// TIA Portal V18 program export: 0 tag tables, 0 data types, 166 data blocks, 119 code blocks (in call order from the OBs), 80 instance data blocks

DATA_BLOCK "GeneralDebug"   // DB1
{ S7_Optimized_Access := 'TRUE' }
// stored: MemoryReserve 100
   VAR
      Debug : Array[1..99] of Bool;
   END_VAR
BEGIN
END_DATA_BLOCK

DATA_BLOCK "DB_Commissioning"   // DB32767
{ S7_Optimized_Access := 'TRUE' }
// stored: AutoNumber false, MemoryReserve 100
   VAR RETAIN
      str : Array[1..8] of String[60];
      bit : Array[1..8] of Bool;
   END_VAR
BEGIN
   str[1] := 'LE4B171420124M33700000131950710';
END_DATA_BLOCK

DATA_BLOCK "DiagnosticDataBlock"   // DB3001
{ S7_Optimized_Access := 'FALSE' }
// stored: AutoNumber false
   VAR RETAIN
      DP : Struct
         DPReadStatus : Int;
         Status : Array[0..1023] of Bool;
      END_STRUCT;
      Profinet : Struct
         PNReadStatus : Int;
         Status : Array[0..1023] of Bool;
      END_STRUCT;
   END_VAR
BEGIN
   // DP.Status[0] : PLC-CPU
   // DP.Status[1] : Remote IO/ET200SP
   // DP.Status[2] : Festo Bus Coupler/总线耦合器
   // DP.Status[3] : CC-LINK
   // DP.Status[4] : Keyence Safety PLC
   // DP.Status[5] : Robot
   // DP.Status[6] : Keyence Laszer
   // DP.Status[7] : Balluff RFID
   // Profinet.Status[0] : ST70&ST80.PLC_CPU
   // Profinet.Status[1] : ST70&ST80.RFID
   // Profinet.Status[2] : ST70.Valves
   // Profinet.Status[3] : ST80.FCPN
   // Profinet.Status[4] : ST70.FCPN
   // Profinet.Status[5] : ST70.Screw
   // Profinet.Status[6] : CMMT-AS
   // Profinet.Status[7] : ST80.Screw
   // Profinet.Status[8] : ST80.Valves
END_DATA_BLOCK

DATA_BLOCK "Sys"   // DB3000
{ S7_Optimized_Access := 'FALSE' }
// stored: AutoNumber false
   VAR RETAIN
      COM : Struct   // Common
         AlwaysOFF : Bool := FALSE;
         AlwaysON : Bool := TRUE;
         FlashTime100mS : Bool := TRUE;   // Hardware Clock Memory 0.1S
         FlashTime200mS : Bool := TRUE;   // Hardware Clock Memory 0.2S
         FlashTime500mS : Bool := FALSE;   // Hardware Clock Memory 0.5S
         FlashTime1S : Bool := FALSE;   // Hardware Clock Memory 1S
         FlashTime2S : Bool := TRUE;   // Hardware Clock Memory 2S
         SpareBit : Bool := FALSE;
         PLCRestarted : Bool := TRUE;
      END_STRUCT;
      SpareB1 : Array[0..7] of Byte;
      DateTime : Struct   // DBX10.0
         Set : Date_And_Time := DT#1990-01-01-00:00:00;
         Read : Date_And_Time := DT#2025-03-12-08:03:05.785;
         Trigger : Bool := FALSE;   // Set
         ReturnValueRead : Int := 0;
         ReturnValueSet : Int := 0;
      END_STRUCT;
      SpareB2 : Array[0..17] of Byte;
      ScanTime : Struct   // DBX50.0
         CyclePrevious : Int := 14;
         CycleMax : Int := 23;
         CycleMin : Int := 9;
      END_STRUCT;
      RETVALI : Int := 0;
      RETVALW : Word := 16#0000;
      VersionManagement : Struct
         ProductLineName : String := 'Assembly Line';
         ProjectNumber : String[20] := 'SZ23055';
         "PLC IP Addr" : Array[0..3] of UInt;
         "HMI IP Addr" : Array[0..3] of UInt;
         PLCVersion : Array[0..1] of UInt;
         HMIVersion : Array[0..1] of UInt;
         "TIA Version" : String := 'TIA V18';
         StationID : Int := 10;
         HMIPageID : Int := 0;
      END_STRUCT;
   END_VAR
BEGIN
   SpareB1[0..7] := 16#00;
   SpareB2[0..17] := 16#00;
   VersionManagement."PLC IP Addr"[0] := 192;
   VersionManagement."PLC IP Addr"[1] := 168;
   VersionManagement."PLC IP Addr"[2..3] := 10;
   VersionManagement."HMI IP Addr"[0] := 192;
   VersionManagement."HMI IP Addr"[1] := 168;
   VersionManagement."HMI IP Addr"[2] := 45;
   VersionManagement."HMI IP Addr"[3] := 11;
   VersionManagement.PLCVersion[0] := 1;
   VersionManagement.PLCVersion[1] := 0;
   VersionManagement.HMIVersion[0] := 1;
   VersionManagement.HMIVersion[1] := 0;
END_DATA_BLOCK

DATA_BLOCK "ST10_GeneralData"   // DB1059
{ S7_Optimized_Access := 'FALSE' }
// stored: AutoNumber false
   VAR
      P_Plus : Array[0..50] of Bool;   // 脉冲沿信号使用Bool,使用需加注释
      ByPass : Array[0..10] of Bool;   // 屏蔽信号,使用需加注释
      HMI : Struct
         AREAPOINTER : Struct
            COORDINATION : Array[1..16] of Bool;
            USER_VERSION : Word;
            SCREEN_NUMBER : Struct
               SCREENTYPE : Int;
               SCREENNUMBER : Int;
               SPARE_1 : Int;
               FIELDNUMBER : Int;
               SPARE_2 : Int;
            END_STRUCT;
            JOB_MAILBOX : Struct
               JOBNUMBER : Int;
               PARAMETER_1 : Int;
               PARAMETER_2 : Int;
               PARAMETER_3 : Int;
            END_STRUCT;
            DATE_TIME_OP : Array[1..12] of Byte;
            DATE_TIME_PLC : Array[1..12] of Byte;
            SPARE : Array[1..22] of Byte;
            DataRecord : Struct   // 数据记录
               RecipeNummer : Word;
               DataRecordNummer : Word;
               Reserve : Word;
               TransferStatus : Word;   // 0,允许传送；2正在传送；4传送已完成，没有错误；12传送完成，出现错误
               Reserve_1 : Word;
            END_STRUCT;
         END_STRUCT;
         Win : Struct   // 弹窗相关变量
            Win : Int;
            WinBullfer : Int;
            "10x弹窗" : Array[1..10] of Int;
            "20x弹窗" : Array[1..10] of Int;
            "30x弹窗" : Array[1..10] of Int;
            "40x弹窗" : Array[1..10] of Int;
            TON : Array[1..40] of TON_TIME;
            "INT" { S7_SetPoint := 'True'} : Array[1..40] of Int;
            "Bool" : Array[1..40] of Bool;
         END_STRUCT;
         StationLightPB : Bool;   // 设备照明按钮
      END_STRUCT;
      Operator : Struct   // 操作员信息
         "Name" : String;   // 姓名
         ID : String;   // 工号
      END_STRUCT;
      TowerLamp : Struct
         PreReady : Bool;   // 等待托盘/等待人工操作
         PreStart : Bool;   // 人工操作完成（自动站False）
         ProcessingFinish : Bool;   // 加工完了 （单个产品加工完成）下个循环开始复位
         Maintenance : Bool;   // 维护提示（缺料OR保养置位1） 无---Flase
      END_STRUCT;
      FlowPartStatus { S7_SetPoint := 'True'} : Array[1..32] of Int;
      FunctionDeSelect : Struct   // 功能屏蔽选择
         "A" : Struct   // 单站屏蔽
            DeSelectPB_Servo380A1 : Bool;
            FunctionDeSelected_Servo380A1 : Bool;
            DeSelectPB_Servo381A1 : Bool;
            FunctionDeSelected_Servo381A1 : Bool;
            DeSelectPB_Servo383A1 : Bool;
            FunctionDeSelected_Servo383A1 : Bool;
            DeSelectPB_Reader800A1 : Bool;
            FunctionDeSelected_Reader800A1 : Bool;
            DeSelectPB_Reader801A1 : Bool;
            FunctionDeSelected_Reader801A1 : Bool;
            DeSelectPB_Reader802A1 : Bool;
            FunctionDeSelected_Reader802A1 : Bool;
            DeSelectPB_Reader803A1 : Bool;
            FunctionDeSelected_Reader803A1 : Bool;
            DeSelectPB_Reader804A1 : Bool;
            FunctionDeSelected_Reader804A1 : Bool;
         END_STRUCT;
         "B" : Struct   // RFID屏蔽
            DeSelectPB_Press372A1 : Bool;
            FunctionDeSelected_Press372A1 : Bool;
            DeSelectPB_Press375A1 : Bool;
            FunctionDeSelected_Press375A1 : Bool;
            DeSelectPB_Reader806A1 : Bool;
            FunctionDeSelected_Reader806A1 : Bool;
            DeSelectPB_TestPress372A1 : Bool;
            FunctionDeSelected_TestPress372A1 : Bool;
            DeSelectPB_TestPress375A1 : Bool;
            FunctionDeSelected_TestPress375A1 : Bool;
         END_STRUCT;
         C : Struct   // 扫码枪屏蔽
            DeSelectPB_Servo382A1 : Bool;
            FunctionDeSelected_Servo382A1 : Bool;
            DeSelectPB_ServoIAI : Bool;
            FunctionDeSelected_ServoIAI : Bool;
            DeSelectPB_IV3810A1 : Bool;
            FunctionDeSelected_IV3810A1 : Bool;
            DeSelectPB_IV3811A1 : Bool;
            FunctionDeSelected_IV3811A1 : Bool;
            DeSelectPB_Glue : Bool;
            FunctionDeSelected_Glue : Bool;
         END_STRUCT;
         "E" : Struct   // 注油屏蔽
            DeSelectPB : Bool;
            FunctionDeSelected : Bool;
         END_STRUCT;
         F : Struct   // 螺丝枪屏蔽
            DeSelectPB_Reader805A1 : Bool;
            FunctionDeSelected_Reader805A1 : Bool;
         END_STRUCT;
         H : Struct   // 油漆笔屏蔽
            DeSelectPB : Bool;
            FunctionDeSelected : Bool;
         END_STRUCT;
         J : Struct   // 油漆笔屏蔽
            DeSelectPB : Bool;
            FunctionDeSelected : Bool;
         END_STRUCT;
         K : Struct   // 油漆笔屏蔽
            DeSelectPB : Bool;
            FunctionDeSelected : Bool;
         END_STRUCT;
         L : Struct   // 油漆笔屏蔽
            DeSelectPB : Bool;
            FunctionDeSelected : Bool;
         END_STRUCT;
         MES : Struct   // MES屏蔽
            DeSelectPB : Bool;
            FunctionDeSelected : Bool;
         END_STRUCT;
         Global : Struct
            DeSelectPB_DryMode : Bool;
            FunctionDeSelected_DryMode : Bool;
            DeSelectPB_ScanFixture : Bool;
            FunctionDeSelected_ScanFixture : Bool;
            Spare_2 : Bool;
            Spare_3 : Bool;
            Spare_4 : Bool;
            Spare_5 : Bool;
            Spare_6 : Bool;
            Spare_7 : Bool;
            Spare_8 : Bool;
            Spare_9 : Bool;
            Spare_10 : Bool;
            Spare_11 : Bool;
            Spare_12 : Bool;
            Spare_13 : Bool;
         END_STRUCT;
      END_STRUCT;
      FlowControl_Handshake : Array[1..32] of Struct   // 流程控制的互锁
         PartPresent : Bool;
         initi : Bool;   // 初始化
         Start : Bool;
         Running : Bool;
         Done : Bool;
         Bypass : Bool;
      END_STRUCT;
      FixtureIDCheck { S7_SetPoint := 'True'} : Array[1..16] of "FixtureCheck_UDT";   // 工装匹配
      ProcessData { S7_SetPoint := 'True'} : Array[0..5] of "ProcessData";
   END_VAR
BEGIN
   // FlowControl_Handshake[2].Bypass : 流程NG
   // FlowControl_Handshake[1] : 主加工流程控制的互锁
   // FlowControl_Handshake[2] : 打标流程控制的互锁
   // FlowControl_Handshake[3] : 产品定位流程控制的互锁
   // FlowControl_Handshake[4] : 贴标流程控制互锁
END_DATA_BLOCK

DATA_BLOCK "Station_Sys"   // DB1060
TITLE = Station system DB
{ S7_Optimized_Access := 'FALSE' }
AUTHOR : RCS
FAMILY : Sys
VERSION : 2.0
// update 20160218
// stored: AutoNumber false
   VAR RETAIN
      ScreenNo : Int;   // For change HMI screen
      SpareB01 : Array[0..7] of Byte;   // *******************************************************************************
      Status : "RCS_SysStatus_V1";   // DBX10.0
      Input : Struct   // DBX20.0 For change PLC I input to PLC inside bit
         OP1 : Struct
            "Function 1" : Bool;
            "Function 2" : Bool;
            "Function 3" : Bool;
            "Function 4" : Bool;
            "Function 5" : Bool;
            "Function 6" : Bool;
            "Function 7" : Bool;
            "Function 8" : Bool;
         END_STRUCT;
         OP2 : Struct
            "Function 1" : Bool;
            "Function 2" : Bool;
            "Function 3" : Bool;
         END_STRUCT;
         OP3 : Struct
            "Function 1" : Bool;
            "Function 2" : Bool;
            "Function 3" : Bool;
         END_STRUCT;
      END_STRUCT;
      SpareB02 : Array[0..13] of Byte;   // *******************************************************************************
      HMI : Struct   // DBX40.0 HMI relation
         AP : Struct   // Area Pointer struct
            S1 : Int;
            CurrentScreenID : Int;
            S3 : Int;
            S4 : Int;
            S5 : Int;
         END_STRUCT;
      END_STRUCT;
      Cmd : "RCS_SysCmd_V1";   // DBX50.0
      SpareB03 : Array[0..7] of Byte;   // *******************************************************************************
      Interface : "RCS_SysComInterface_V1";   // DBX60.0
      SpareB04 : Array[0..3] of Byte;   // *******************************************************************************
      Initial : Struct   // DBX70.0
         Set : Bool;   // Trigger by HMI Button,[0]Total trigger
         Running : Bool;   // [0]Total initial Running
         OK : Bool;   // finish
      END_STRUCT;
      SpareB05 : Array[0..27] of Byte;   // *******************************************************************************
      Auto : "RCS_SysAuto_V1";   // DBX100.0
      SpareB10 : Array[0..5] of Byte;   // *******************************************************************************
      "A" : Struct   // DBX110.0 Auto control bit for some device
         "Device1 Auto control" : Bool;
         "Device2 Auto control" : Bool;
         "Device3 Auto control" : Bool;
         "Device4 Auto control" : Bool;
         "Device 01" : Struct
            "Function 1" : Bool;   // Flash
            "Function 2" : Bool;
            "Function 3" : Bool;   // Flash
         END_STRUCT;
         "Device 02" : Struct
            "Function 1" : Bool;   // Flash
            "Function 2" : Bool;
            "Function 3" : Bool;   // Flash
         END_STRUCT;
      END_STRUCT;
      SpareB11 : Array[0..33] of Byte;   // *******************************************************************************
      Manual : "RCS_SysManual_V1";   // DBX150.0
      SpareB12 : Array[0..6] of Byte;   // *******************************************************************************
      "M" : Struct   // DBX160.0 Manual control bit for some device
         "Device1 Manual control" : Bool;
         "Device2 Manual control" : Bool;
         "Device3 Manual control" : Bool;
         "Device4 Manual control" : Bool;
      END_STRUCT;
      SpareB13 : Array[0..37] of Byte;   // *******************************************************************************
      Safety : "RCS_SysSafety_V1";   // DBX200.0
      SpareB20 : Array[0..9] of Byte;   // *******************************************************************************
      Signal : Struct   // DBX220.0
         MainPressureSwitch1 : Bool;
         MainPressureSwitch2 : Bool;
         MainPressureSwitch3 : Bool;
      END_STRUCT;
      SpareB21 : Array[0..36] of Byte;   // *******************************************************************************
      Flag : Struct   // DBX260.0
         Processstart : Bool;
         PeocessComplete : Bool;
         IndexTable : Struct
            Interlock : Bool;
            TableRunning : Bool;   // Complete cycle Running
            StopandPosition : Bool;
            PositionOK : Bool;
            PositionNG : Bool;
            FixtureOK : Bool;
            FixtureNG : Bool;
            InitialOK : Bool;
         END_STRUCT;
      END_STRUCT;
      SpareB22 : Array[0..5] of Byte;   // *******************************************************************************
      P : Struct   // Positive RLO Edge Detection:-(P)- DBX270
         Record : Bool;
         "Set index run" : Bool;
         initial : Array[0..7] of Bool;
      END_STRUCT;
      SpareB23 : Array[0..5] of Byte;   // *******************************************************************************
      N : Struct   // Negative RLO Edge Detection:-(N)- DBX280
         Spare : Bool;
      END_STRUCT;
      SpareB24 : Array[0..17] of Byte;   // *******************************************************************************
      Alarm : "RCS_SysAlarmWarning_V1";   // DBX300.0
      SpareB30 : Array[0..7] of Byte;   // *******************************************************************************
      Warning : "RCS_SysAlarmWarning_V1";   // DBX310.0 / DBX500.0
      SpareB31 : Array[0..7] of Byte;   // *******************************************************************************
      AlarmTimes : Struct   // DBX320 If a fault continue happened over Limit times, than Auto running will be stopped / If a fault continue happened over Limit_times，Auto running will be stopped
         ForceStop : Bool;   // DBX320.0 / DBX650.0
         Reset : Bool;
         Limit : Int;
      END_STRUCT;
      SpareB33 : Array[0..5] of Byte;   // *******************************************************************************
      AlarmWarning : Int;   // DBX330 1:Alarm 2:Warning / DBX660 1:Alarm 2:Warning
      SpareB34 : Array[0..17] of Byte;   // *******************************************************************************
      Count : "RCS_SysCount_V1";   // DBX350.0 / DBX700.0
      SpareB40 : Array[0..11] of Byte;   // *******************************************************************************
      TotalCycleTime : "RCS_SysCycleTime_V1";   // DBX500.0 / DBX850.0
      SpareB41 : Array[0..11] of Byte;   // *******************************************************************************
      MachineCycleTime : "RCS_SysCycleTime_V1";   // DBX600.0 / DBX950.0
      SpareB42 : Array[0..11] of Byte;   // *******************************************************************************
      UserName { S7_SetPoint := 'True'} : String[20];   // DBX700.0
   END_VAR
BEGIN
   // Cmd.Record : 记录
   // Cmd.BuzzerOn : 蜂鸣器 On
   Cmd.OnOffLine := TRUE;
END_DATA_BLOCK

DATA_BLOCK "ST10_SysInput"   // DB1001
{ S7_Optimized_Access := 'TRUE' }
// stored: AutoNumber false, MemoryReserve 100
   VAR
      HMI_Button : Struct
         ControlOn : Bool := false;   // HMI_上电按钮
         ControlOff : Bool;   // HMI_断电按钮
         MachineStart : Bool := false;   // HMI_设备启动按钮
         MachineStop : Bool := false;   // HMI_设备停止按钮
         ResetButton : Bool := false;   // HMI_复位按钮
         "Manual/Auto" : Bool := false;   // HMI_手/自动切换按钮
         SafetyGateUnlock : Bool := false;   // HMI_安全门解锁按钮
         "E-Stop" : Bool := false;   // HMI_急停
      END_STRUCT;
      Sys : Struct
         iCircuitBreakerOK1 : Bool;   // 电子断路器 OK
         iCircuitBreakerOK2 : Bool;
         iPressure : Bool;   // 气压监控
      END_STRUCT;
      "iE-StopPB" : Array[1..20] of Bool;   // 急停按钮PB
      iSafetyGatFeedBack : Array[1..20] of Bool;   // 安全门
      iSafetydoorLockingFeedBack : Array[1..20] of Bool;   // 安全门反馈
      iMaterieldoorLockingFeedBack : Array[1..20] of Bool;   // 安全门反馈
   END_VAR
BEGIN
END_DATA_BLOCK

DATA_BLOCK "ST10_SysOutput"   // DB1002
{ S7_Optimized_Access := 'TRUE' }
// stored: AutoNumber false, MemoryReserve 100
   VAR
      oTowerLight : Struct
         Red : Bool;
         Yellow : Bool;
         Green : Bool;
         Blue : Bool;
      END_STRUCT;
      HMIButtonLight : Struct
         ControlOn : Bool := false;   // HMI_上电按钮
         ControlOff : Bool;   // HMI_断电按钮
         MachineStart : Bool := false;   // HMI_设备启动按钮
         MachineStop : Bool := false;   // HMI_设备停止按钮
         ResetButton : Bool := false;   // HMI_复位按钮
         "Manual/Auto" : Bool := false;   // HMI_手/自动切换按钮
         SafetyGateUnlock : Bool := false;   // HMI_安全门解锁按钮
      END_STRUCT;
      BoxLight : Struct
         oMachineStartLight : Bool;   // 启动按钮PB
         oMachineStopLight : Bool;   // 停止按钮PB
         oResetLight : Bool;   // 复位按钮PB
         oSafetyGateUnlockLight : Bool;   // 安全门解锁按钮PB
      END_STRUCT;
      SafetyDoorCoil : Array[1..20] of Bool;
      MaterialDoorCoil : Array[1..20] of Bool;
   END_VAR
BEGIN
END_DATA_BLOCK

DATA_BLOCK "AutoProcessControl"   // DB5100
{ S7_Optimized_Access := 'FALSE' }
// stored: AutoNumber false
   VAR
      A_Table_1Scan : Struct   // 自动页面
         Robot1PickPrimit : Bool;
         Spare_2 : Bool;
         Spare_3 : Bool;
         Spare_4 : Bool;
         Spare_5 : Bool;
         Spare_6 : Bool;
         Spare_7 : Bool;
         Spare_8 : Bool;
         Spare_9 : Bool;
         Spare_10 : Bool;
         Spare_11 : Bool;
         Spare_12 : Bool;
         Spare_13 : Bool;
         Spare_14 : Bool;
         Spare_15 : Bool;
         Spare_16 : Bool;
      END_STRUCT;
      A_Table_1Loading : Struct
         Robot1PickPrimit : Bool;
         Spare_2 : Bool;
         Spare_3 : Bool;
         Spare_4 : Bool;
         Spare_5 : Bool;
         Spare_6 : Bool;
         Spare_7 : Bool;
         Spare_8 : Bool;
         Spare_9 : Bool;
         Spare_10 : Bool;
         Spare_11 : Bool;
         Spare_12 : Bool;
         Spare_13 : Bool;
         Spare_14 : Bool;
         Spare_15 : Bool;
         Spare_16 : Bool;
         ServoRunCount : Int;
      END_STRUCT;
      A_Table_2Scan : Struct
         Robot3PickPrimit : Bool;
         Spare_2 : Bool;
         Spare_3 : Bool;
         Spare_4 : Bool;
         Spare_5 : Bool;
         Spare_6 : Bool;
         Spare_7 : Bool;
         Spare_8 : Bool;
         Spare_9 : Bool;
         Spare_10 : Bool;
         Spare_11 : Bool;
         Spare_12 : Bool;
         Spare_13 : Bool;
         Spare_14 : Bool;
         Spare_15 : Bool;
         Spare_16 : Bool;
      END_STRUCT;
      A_Table_2Loading : Struct
         Robot3PickPrimit : Bool;
         Spare_2 : Bool;
         Spare_3 : Bool;
         Spare_4 : Bool;
         Spare_5 : Bool;
         Spare_6 : Bool;
         Spare_7 : Bool;
         Spare_8 : Bool;
         Spare_9 : Bool;
         Spare_10 : Bool;
         Spare_11 : Bool;
         Spare_12 : Bool;
         Spare_13 : Bool;
         Spare_14 : Bool;
         Spare_15 : Bool;
         Spare_16 : Bool;
         ServoRunCount : Int;
      END_STRUCT;
      A_ScanRotary : Struct
         Robot1PickPrimit : Bool;
         Robot1PutPrimit : Bool;
         Spare_3 : Bool;
         Spare_4 : Bool;
         Spare_5 : Bool;
         Spare_6 : Bool;
         Spare_7 : Bool;
         Spare_8 : Bool;
         Spare_9 : Bool;
         Spare_10 : Bool;
         Spare_11 : Bool;
         Spare_12 : Bool;
         Spare_13 : Bool;
         Spare_14 : Bool;
         Spare_15 : Bool;
         Spare_16 : Bool;
      END_STRUCT;
      B_Press_1 : Struct   // 自动页面
         Robot1PickPrimit : Bool;
         Robot1PutShaftPrimit : Bool;
         Robot1PutRingPrimit : Bool;
         Spare_4 : Bool;
         Spare_5 : Bool;
         Spare_6 : Bool;
         Spare_7 : Bool;
         Spare_8 : Bool;
         Spare_9 : Bool;
         Spare_10 : Bool;
         Spare_11 : Bool;
         Spare_12 : Bool;
         Spare_13 : Bool;
         Spare_14 : Bool;
         Spare_15 : Bool;
         Spare_16 : Bool;
         GripStatus : Int;
      END_STRUCT;
      B_Press_2 : Struct
         Robot3PickPrimit : Bool;
         Robot3PutRingPrimit : Bool;
         Robot2PutPrimit : Bool;
         Spare_4 : Bool;
         Spare_5 : Bool;
         Spare_6 : Bool;
         Spare_7 : Bool;
         Spare_8 : Bool;
         Spare_9 : Bool;
         Spare_10 : Bool;
         Spare_11 : Bool;
         Spare_12 : Bool;
         Spare_13 : Bool;
         Spare_14 : Bool;
         Spare_15 : Bool;
         Spare_16 : Bool;
         GripStatus : Int;
      END_STRUCT;
      C_Glue : Struct
         Robot2PickPrimit : Bool;
         Robot1PutPrimit : Bool;
         Robot2MaganePutPrimit : Bool;
         Spare_4 : Bool;
         Spare_5 : Bool;
         Spare_6 : Bool;
         Spare_7 : Bool;
         Spare_8 : Bool;
         GlueTest : Bool;
         Spare_10 : Bool;
         Spare_11 : Bool;
         Spare_12 : Bool;
         Spare_13 : Bool;
         Spare_14 : Bool;
         Spare_15 : Bool;
         Spare_16 : Bool;
      END_STRUCT;
      H_ShafeLine : Struct
         Robot1PickPrimit : Bool;
         Spare_2 : Bool;
         Spare_3 : Bool;
         Spare_4 : Bool;
         Spare_5 : Bool;
         Spare_6 : Bool;
         Spare_7 : Bool;
         Spare_8 : Bool;
         EmptyMaterial : Bool;   // 托盘清料反转
         LineTest : Bool;
         Spare_11 : Bool;
         Spare_12 : Bool;
         Spare_13 : Bool;
         Spare_14 : Bool;
         Spare_15 : Bool;
         Spare_16 : Bool;
      END_STRUCT;
      J_MagnetLine : Struct
         Robot2PickPrimit : Bool;
         Spare_2 : Bool;
         Spare_3 : Bool;
         Spare_4 : Bool;
         Spare_5 : Bool;
         Spare_6 : Bool;
         Spare_7 : Bool;
         Spare_8 : Bool;
         EmptyMaterial : Bool;   // 托盘清料反转
         LineTest : Bool;
         Spare_11 : Bool;
         Spare_12 : Bool;
         Spare_13 : Bool;
         Spare_14 : Bool;
         Spare_15 : Bool;
         Spare_16 : Bool;
      END_STRUCT;
      K_ShafeLine : Struct
         Robot2PickPrimit : Bool;
         Spare_2 : Bool;
         Spare_3 : Bool;
         Spare_4 : Bool;
         Spare_5 : Bool;
         Spare_6 : Bool;
         Spare_7 : Bool;
         Spare_8 : Bool;
         EmptyMaterial : Bool;   // 托盘清料反转
         LineTest : Bool;
         Spare_11 : Bool;
         Spare_12 : Bool;
         Spare_13 : Bool;
         Spare_14 : Bool;
         Spare_15 : Bool;
         Spare_16 : Bool;
      END_STRUCT;
      L_ShafeLine : Struct
         Robot3PutPrimit : Bool;
         Spare_2 : Bool;
         Spare_3 : Bool;
         Spare_4 : Bool;
         Spare_5 : Bool;
         Spare_6 : Bool;
         Spare_7 : Bool;
         Spare_8 : Bool;
         EmptyMaterial : Bool;   // 托盘清料反转
         LineTest : Bool;
         Spare_11 : Bool;
         Spare_12 : Bool;
         Spare_13 : Bool;
         Spare_14 : Bool;
         Spare_15 : Bool;
         Spare_16 : Bool;
      END_STRUCT;
      Headt : Struct
         PalletUnloadingPrimit : Bool;
         Spare_2 : Bool;
         Spare_3 : Bool;
         Spare_4 : Bool;
         Spare_5 : Bool;
         Spare_6 : Bool;
         Spare_7 : Bool;
         Spare_8 : Bool;
         Spare_9 : Bool;
         Spare_10 : Bool;
         Spare_11 : Bool;
         Spare_12 : Bool;
         Spare_13 : Bool;
         Spare_14 : Bool;
         Spare_15 : Bool;
         Spare_16 : Bool;
      END_STRUCT;
      Robot2ScanNG : Struct
         PutPrimit : Bool;
         Spare_2 : Bool;
         Spare_3 : Bool;
         Spare_4 : Bool;
         Spare_5 : Bool;
         Spare_6 : Bool;
         Spare_7 : Bool;
         Spare_8 : Bool;
         Spare_9 : Bool;
         Spare_10 : Bool;
         Spare_11 : Bool;
         Spare_12 : Bool;
         Spare_13 : Bool;
         Spare_14 : Bool;
         Spare_15 : Bool;
         Spare_16 : Bool;
      END_STRUCT;
      Robot2GlueNG : Struct
         PutPrimit : Bool;
         Spare_2 : Bool;
         Spare_3 : Bool;
         Spare_4 : Bool;
         Spare_5 : Bool;
         Spare_6 : Bool;
         Spare_7 : Bool;
         Spare_8 : Bool;
         Spare_9 : Bool;
         Spare_10 : Bool;
         Spare_11 : Bool;
         Spare_12 : Bool;
         Spare_13 : Bool;
         Spare_14 : Bool;
         Spare_15 : Bool;
         Spare_16 : Bool;
      END_STRUCT;
      NG_1 : Struct
         Robot1PutPrimit_1 : Bool;
         Robot1PutPrimit_2 : Bool;
         Robot1PutPrimit_3 : Bool;
         Spare_4 : Bool;
         Spare_5 : Bool;
         Spare_6 : Bool;
         Spare_7 : Bool;
         Spare_8 : Bool;
         DoorRequest : Bool;
         Spare_10 : Bool;
         Spare_11 : Bool;
         Spare_12 : Bool;
         Spare_13 : Bool;
         Spare_14 : Bool;
         Spare_15 : Bool;
         Spare_16 : Bool;
      END_STRUCT;
      NG_2 : Struct
         Robot3PutPrimit_1 : Bool;
         Robot3PutPrimit_2 : Bool;
         Robot3PutPrimit_3 : Bool;
         Spare_4 : Bool;
         Spare_5 : Bool;
         Spare_6 : Bool;
         Spare_7 : Bool;
         Spare_8 : Bool;
         DoorRequest : Bool;
         Spare_10 : Bool;
         Spare_11 : Bool;
         Spare_12 : Bool;
         Spare_13 : Bool;
         Spare_14 : Bool;
         Spare_15 : Bool;
         Spare_16 : Bool;
      END_STRUCT;
      NGBuffer : Struct
         Robot3PPickMagnetNGPrimit : Bool;
         PickGlueNGPrimit : Bool;
         Spare_17 : Bool;
         Spare_4 : Bool;
         Spare_5 : Bool;
         Spare_6 : Bool;
         Spare_7 : Bool;
         Spare_8 : Bool;
         Spare_9 : Bool;
         Spare_10 : Bool;
         Spare_11 : Bool;
         Spare_12 : Bool;
         Spare_13 : Bool;
         Spare_14 : Bool;
         Spare_15 : Bool;
         Spare_16 : Bool;
      END_STRUCT;
      Fixture1Code : Struct
         Robot1CodeReadReq : Bool;
         Spare_17 : Bool;
         Spare_18 : Bool;
         Spare_4 : Bool;
         Spare_5 : Bool;
         Spare_6 : Bool;
         Spare_7 : Bool;
         Spare_8 : Bool;
         Spare_9 : Bool;
         Spare_10 : Bool;
         Spare_11 : Bool;
         Spare_12 : Bool;
         Spare_13 : Bool;
         Spare_14 : Bool;
         Spare_15 : Bool;
         Spare_16 : Bool;
      END_STRUCT;
      Fixture2Code : Struct
         Robot3CodeReadReq : Bool;
         Spare_17 : Bool;
         Spare_18 : Bool;
         Spare_4 : Bool;
         Spare_5 : Bool;
         Spare_6 : Bool;
         Spare_7 : Bool;
         Spare_8 : Bool;
         Spare_9 : Bool;
         Spare_10 : Bool;
         Spare_11 : Bool;
         Spare_12 : Bool;
         Spare_13 : Bool;
         Spare_14 : Bool;
         Spare_15 : Bool;
         Spare_16 : Bool;
      END_STRUCT;
      Robot_1 : Struct
         GluePutFlag : Bool;
         NGPutFlag : Bool;
         MaintenanceRequest : Bool;
         HomeRequest : Bool;
         Spare_5 : Bool;
         Spare_6 : Bool;
         Spare_7 : Bool;
         Spare_8 : Bool;
         ReadyToRobot2 : Bool;
         ClearPart : Bool;
         GripScanRequest : Bool;
         OnePart : Bool;
         Spare_13 : Bool;
         Spare_14 : Bool;
         Spare_15 : Bool;
         Spare_16 : Bool;
      END_STRUCT;
      Robot_2 : Struct
         PalletPickFlag : Bool;
         MagnetScanFlag : Bool;
         GluePutFlag : Bool;
         GluePickFlag : Bool;
         Press2PutFlag : Bool;
         GlueNGPutFlag : Bool;
         ScanNGPutFlag : Bool;
         Spare_8 : Bool;
         ReadyToRobot1 : Bool;
         ReadyToRobot3 : Bool;
         MaintenanceRequest : Bool;
         HomeRequest : Bool;
         GripScanRequest : Bool;
         Spare_14 : Bool;
         Spare_15 : Bool;
         Spare_16 : Bool;
      END_STRUCT;
      Robot_3 : Struct
         Press2PutFlag : Bool;
         Press2PickFlag : Bool;
         GlueNGPickFlag : Bool;
         ScanNGPickFlag : Bool;
         NGPutFlag : Bool;
         Spare_10 : Bool;
         Spare_9 : Bool;
         Spare_8 : Bool;
         ReadyToRobot2 : Bool;
         PalletFull : Bool;
         MaintenanceRequest : Bool;
         HomeRequest : Bool;
         GripScanRequest : Bool;
         Spare_14 : Bool;
         Spare_15 : Bool;
         Spare_16 : Bool;
      END_STRUCT;
      Global : Struct
         H : Struct
            EmptyPallet : Bool;
            LoadStopRequestPallet_1 : Bool;
            LoadStopRequestPallet_2 : Bool;
            LoadStopRequestPallet_3 : Bool;
            LoadStopRequestPallet_4 : Bool;
            EmptyStopRequestPallet_1 : Bool;
            EmptyStopRequestPallet_2 : Bool;
            EmptyStopRequestPallet_3 : Bool;
            Spare : Bool;
            Spare_1 : Bool;
            Spare_2 : Bool;
            Spare_3 : Bool;
            Spare_4 : Bool;
            Spare_5 : Bool;
            Spare_6 : Bool;
            Spare_7 : Bool;
         END_STRUCT;
         J : Struct
            EmptyPallet : Bool;
            LoadStopRequestPallet_1 : Bool;
            LoadStopRequestPallet_2 : Bool;
            LoadStopRequestPallet_3 : Bool;
            LoadStopRequestPallet_4 : Bool;
            EmptyStopRequestPallet_1 : Bool;
            EmptyStopRequestPallet_2 : Bool;
            EmptyStopRequestPallet_3 : Bool;
            Spare : Bool;
            Spare_1 : Bool;
            Spare_2 : Bool;
            Spare_3 : Bool;
            Spare_4 : Bool;
            Spare_5 : Bool;
            Spare_6 : Bool;
            Spare_7 : Bool;
         END_STRUCT;
         K : Struct
            EmptyPallet : Bool;
            LoadStopRequestPallet_1 : Bool;
            LoadStopRequestPallet_2 : Bool;
            LoadStopRequestPallet_3 : Bool;
            LoadStopRequestPallet_4 : Bool;
            EmptyStopRequestPallet_1 : Bool;
            EmptyStopRequestPallet_2 : Bool;
            EmptyStopRequestPallet_3 : Bool;
            Spare : Bool;
            Spare_1 : Bool;
            Spare_2 : Bool;
            Spare_3 : Bool;
            Spare_4 : Bool;
            Spare_5 : Bool;
            Spare_6 : Bool;
            Spare_7 : Bool;
         END_STRUCT;
         L : Struct
            EmptyPallet : Bool;
            LoadStopRequestPallet_1 : Bool;
            LoadStopRequestPallet_2 : Bool;
            LoadStopRequestPallet_3 : Bool;
            LoadStopRequestPallet_4 : Bool;
            EmptyStopRequestPallet_1 : Bool;
            EmptyStopRequestPallet_2 : Bool;
            EmptyStopRequestPallet_3 : Bool;
            Spare : Bool;
            Spare_1 : Bool;
            Spare_2 : Bool;
            Spare_3 : Bool;
            Spare_4 : Bool;
            Spare_5 : Bool;
            Spare_6 : Bool;
            Spare_7 : Bool;
         END_STRUCT;
         H_EmptyPallet : Bool;
         J_EmptyPallet : Bool;
         K_EmptyPallet : Bool;
         L_EmptyPallet : Bool;
         ALL_EmptyPallet : Bool;
         ALL_BeltPalletEmptyFinish : Bool;
         Spare_7 : Bool;
         Spare_8 : Bool;
         Spare_9 : Bool;
         Spare_10 : Bool;
         Spare_11 : Bool;
         Spare_12 : Bool;
         Spare_13 : Bool;
         Spare_14 : Bool;
         Spare_15 : Bool;
         Spare_16 : Bool;
         P : Array[0..60] of Bool;
      END_STRUCT;
      P : Array[0..40] of Bool;
      Status : Struct
         A1TableScan : Struct
            Status : Int;
         END_STRUCT;
         A1TableUnloading : Struct
            Status : Int;
         END_STRUCT;
         A1RotaryScan : Struct
            Status : Int;
         END_STRUCT;
         B1Press : Struct
            Status : Int;
         END_STRUCT;
         FRobot_1 : Struct
            Status : Int;
         END_STRUCT;
         A1FixtureCodeScan : Struct
            Status : Int;
         END_STRUCT;
         CGlueing : Struct
            Status : Int;
         END_STRUCT;
         FRobot_2 : Struct
            Status : Int;
         END_STRUCT;
         A2TableScan : Struct
            Status : Int;
         END_STRUCT;
         A2TableUnloading : Struct
            Status : Int;
         END_STRUCT;
         ChangeOver : Struct
            Status : Int;
         END_STRUCT;
         B2Press : Struct
            Status : Int;
         END_STRUCT;
         FRobot_3 : Struct
            Status : Int;
         END_STRUCT;
         A2FixtureCodeScan : Struct
            Status : Int;
         END_STRUCT;
         HShaftLifting : Struct
            Status : Int;
         END_STRUCT;
         JMagnetLifting : Struct
            Status : Int;
         END_STRUCT;
         KReserveLifting : Struct
            Status : Int;
         END_STRUCT;
         LUnloadingTrans : Struct
            Status : Int;
         END_STRUCT;
         "HShaftLoad&Unload" : Struct
            Status : Int;
         END_STRUCT;
         "JMagnetLoad&Unload" : Struct
            Status : Int;
         END_STRUCT;
         "KReserveLoad&Unload" : Struct
            Status : Int;
         END_STRUCT;
         "LUnloadingLoad&Unload" : Struct
            Status : Int;
         END_STRUCT;
         Solidify : Struct
            Status : Int;
         END_STRUCT;
         ENG_1 : Struct
            Status : Int;
         END_STRUCT;
         ENG_2 : Struct
            Status : Int;
         END_STRUCT;
      END_STRUCT;
   END_VAR
BEGIN
END_DATA_BLOCK

DATA_BLOCK "AutoProcessData"   // DB1600
{ S7_Optimized_Access := 'FALSE' }
// stored: AutoNumber false
   VAR RETAIN
      A_ScanRotate : "ProcessData";
      F_Robot1Grip1 { S7_SetPoint := 'True'} : "ProcessData";
      F_Robot1Grip2 { S7_SetPoint := 'True'} : "ProcessData";
      B_Press1 { S7_SetPoint := 'True'} : "ProcessData";
      C_Glue { S7_SetPoint := 'True'} : "ProcessData";
      F_Robot2Grip1 { S7_SetPoint := 'True'} : "ProcessData";
      F_Robot2Grip2 { S7_SetPoint := 'True'} : "ProcessData";
      C_GlueNGBuffer { S7_SetPoint := 'True'} : "ProcessData";
      C_MagnScanNGBuffer { S7_SetPoint := 'True'} : "ProcessData";
      B_Press2 { S7_SetPoint := 'True'} : "ProcessData";
      F_Robot3Grip1 { S7_SetPoint := 'True'} : "ProcessData";
      F_Robot3Grip2 { S7_SetPoint := 'True'} : "ProcessData";
      H_ShafeLine { S7_SetPoint := 'True'} : "ProcessData";
      J_ShafeLine { S7_SetPoint := 'True'} : "ProcessData";
      K_ShafeLine { S7_SetPoint := 'True'} : "ProcessData";
      L_ShafeLine { S7_SetPoint := 'True'} : "ProcessData";
      ClearData { S7_SetPoint := 'True'} : "ProcessData";
      A_Table_1 { S7_SetPoint := 'True'} : Array[1..10] of "TableProcessData";
      A_Table_2 { S7_SetPoint := 'True'} : Array[1..10] of "TableProcessData";
      FixtureCode_A1 { S7_SetPoint := 'True'} : Array[1..10] of String[128];
      FixtureCode_A2 { S7_SetPoint := 'True'} : Array[1..10] of String[128];
      GlobalData : Struct
         Table1CodeOKFlag : Bool;
         Table2CodeOKFlag : Bool;
         Fixture1CodeOKFlag : Bool;
         Fixture2CodeOKFlag : Bool;
         Robot2GripperCodeOKFlag : Bool;
         Robot1GripperCodeOKFlag : Bool;
         Robot3GripperCodeOKFlag : Bool;
         Spare_8 : Bool;
         Spare_9 : Bool;
         Spare_10 : Bool;
         Spare_11 : Bool;
         Spare_12 : Bool;
         Spare_13 : Bool;
         Spare_14 : Bool;
         Spare_15 : Bool;
         Spare_16 : Bool;
         DataIndex { S7_SetPoint := 'True'} : Int := 1;
         Robot1GripCodeStatus1 : Int;
         Robot1GripCodeStatus2 : Int;
         Robot1GripCodeStatus3 : Int;
         Robot1GripCodeStatus4 : Int;
         Robot2GripCodeStatus1 : Int;
         Robot2GripCodeStatus2 : Int;
         Robot2GripCodeStatus3 : Int;
         Robot2GripCodeStatus4 : Int;
         Robot3GripCodeStatus1 : Int;
         Robot3GripCodeStatus2 : Int;
         Robot3GripCodeStatus3 : Int;
         Robot3GripCodeStatus4 : Int;
         FixtureCode_A1Status1 : Int;
         FixtureCode_A1Status2 : Int;
         FixtureCode_A1Status3 : Int;
         FixtureCode_A1Status4 : Int;
         FixtureCode_A1Status5 : Int;
         FixtureCode_A1Status6 : Int;
         FixtureCode_A1Status7 : Int;
         FixtureCode_A1Status8 : Int;
         FixtureCode_A1Status9 : Int;
         FixtureCode_A1Status10 : Int;
         FixtureCode_A2Status1 : Int;
         FixtureCode_A2Status2 : Int;
         FixtureCode_A2Status3 : Int;
         FixtureCode_A2Status4 : Int;
         FixtureCode_A2Status5 : Int;
         FixtureCode_A2Status6 : Int;
         FixtureCode_A2Status7 : Int;
         FixtureCode_A2Status8 : Int;
         FixtureCode_A2Status9 : Int;
         FixtureCode_A2Status10 : Int;
         Spare : Array[1..332] of Byte;
      END_STRUCT;
      DataBuffer : Array[1..30] of "ProcessData";
      GripperCode_R1 { S7_SetPoint := 'True'} : Array[1..10] of String[128];
      GripperCode_R2 { S7_SetPoint := 'True'} : Array[1..10] of String[128];
      GripperCode_R3 { S7_SetPoint := 'True'} : Array[1..10] of String[128];
   END_VAR
BEGIN
   A_Table_1[1].Code := 'SZ23055-OP010-E-Compressor-ring1 Loading tooling-1';
   A_Table_1[2].Code := 'SZ23055-OP010-E-Compressor-ring1 Loading tooling-2';
   A_Table_2[1].Code := 'SZ23055-OP010-E-Compressor-ring2 Loading tooling-1$R';
END_DATA_BLOCK

DATA_BLOCK "AutoProcessData_Buffer"   // DB1601
{ S7_Optimized_Access := 'FALSE' }
// stored: AutoNumber false
   VAR RETAIN
      DataBuffer : Array[0..55] of "ProcessData";
      DataBuffer_1 : "ProcessData";
      DataBuffer_2 { S7_SetPoint := 'True'} : "ProcessData";
      DataBuffer_3 { S7_SetPoint := 'True'} : "ProcessData";
      DataBuffer_4 { S7_SetPoint := 'True'} : "ProcessData";
      DataBuffer_5 { S7_SetPoint := 'True'} : "ProcessData";
      DataBuffer_6 { S7_SetPoint := 'True'} : "ProcessData";
      VAL { S7_SetPoint := 'True'} : Int;
      SelectButton : Int;
      Button_2 : Bool;
      Button_3 : Bool;
      Button_4 : Bool;
      Button_5 : Bool;
      Button_6 : Bool;
   END_VAR
BEGIN
END_DATA_BLOCK

DATA_BLOCK "AutoProcessData_Buffer_Clear"   // DB1602
{ S7_Optimized_Access := 'FALSE' }
// stored: AutoNumber false
   VAR RETAIN
      DataBuffer : Array[0..60] of "ProcessData";
      DataBufferClear : "ProcessData";
      VAL { S7_SetPoint := 'True'} : Int;
   END_VAR
BEGIN
END_DATA_BLOCK

DATA_BLOCK "PalletRelease"   // DB9001
{ S7_Optimized_Access := 'FALSE' }
// stored: AutoNumber false
   VAR
      Buffer : Struct
         AskPallet : Bool;
         UnloadFlag : Bool;
      END_STRUCT;
      LaserMarking : Struct
         AskPallet : Bool;
         UnloadFlag : Bool;
      END_STRUCT;
      Print : Struct
         AskPallet : Bool;
         UnloadFlag : Bool;
      END_STRUCT;
      Spare : Struct
         AskPallet : Bool;
         UnloadFlag : Bool;
      END_STRUCT;
      Spare2 : Struct
         AskPallet : Bool;
         UnloadFlag : Bool;
      END_STRUCT;
      "Time" : Array[0..1] of TOF_TIME;
      LaserMarkingBuffer : "LaserMarkingBuffer";
   END_VAR
BEGIN
END_DATA_BLOCK

DATA_BLOCK "ST10_PM"   // DB1063
{ S7_Optimized_Access := 'FALSE' }
// stored: AutoNumber false
   VAR RETAIN
      Num : Array[1..32] of "RCS_PMInterface_V1";
      Status { S7_SetPoint := 'True'} : Array[1..50] of Int;
   END_VAR
BEGIN
   // Num[1] : laszer marking
   // Num[2] : LabelFeeder
END_DATA_BLOCK

DATA_BLOCK "TON"   // DB163
{ S7_Optimized_Access := 'TRUE' }
// stored: AutoNumber false, MemoryReserve 100
   VAR
      TON : Array[0..100] of TON_TIME;
      CTU { S7_SetPoint := 'True'} : Array[0..20] of IEC_DCOUNTER;
   END_VAR
   VAR RETAIN
      P { S7_SetPoint := 'True'} : Array[0..20] of Bool;
   END_VAR
BEGIN
END_DATA_BLOCK

DATA_BLOCK "ST10_DeviceError"   // DB1067
{ S7_Optimized_Access := 'FALSE' }
// stored: AutoNumber false
   VAR RETAIN
      CylinderFault : Struct   // Cylinder Error（气缸错误）
         C1GoWorkFault : Bool;   // Cyl1
         C1GoHomeFault : Bool;   // Cyl1
         C1SensorPositionFault : Bool;   // Cyl1
         C1SpareFault : Bool;
         C2GoWorkFault : Bool;   // Cyl2
         C2GoHomeFault : Bool;   // Cyl2
         C2SensorPositionFault : Bool;   // Cyl2
         C2SpareFault : Bool;
         C3GoWorkFault : Bool;   // Cyl3
         C3GoHomeFault : Bool;   // Cyl3
         C3SensorPositionFault : Bool;   // Cyl3
         C3SpareFault : Bool;
         C4GoWorkFault : Bool;   // Cyl4
         C4GoHomeFault : Bool;   // Cyl4
         C4SensorPositionFault : Bool;   // Cyl4
         C4SpareFault : Bool;
         C5GoWorkFault : Bool;   // Cyl5
         C5GoHomeFault : Bool;   // Cyl5
         C5SensorPositionFault : Bool;   // Cyl5
         C5SpareFault : Bool;
         C6GoWorkFault : Bool;   // Cyl6
         C6GoHomeFault : Bool;   // Cyl6
         C6SensorPositionFault : Bool;   // Cyl6
         C6SpareFault : Bool;
         C7GoWorkFault : Bool;   // Cyl7
         C7GoHomeFault : Bool;   // Cyl7
         C7SensorPositionFault : Bool;   // Cyl7
         C7SpareFault : Bool;
         C8GoWorkFault : Bool;   // Cyl8
         C8GoHomeFault : Bool;   // Cyl8
         C8SensorPositionFault : Bool;   // Cyl8
         C8SpareFault : Bool;
         C9GoWorkFault : Bool;   // Cyl9
         C9GoHomeFault : Bool;   // Cyl9
         C9SensorPositionFault : Bool;   // Cyl9
         C9SpareFault : Bool;
         C10GoWorkFault : Bool;   // Cyl10
         C10GoHomeFault : Bool;   // Cyl10
         C10SensorPositionFault : Bool;   // Cyl10
         C10SpareFault : Bool;
         C11GoWorkFault : Bool;   // Cyl11
         C11GoHomeFault : Bool;   // Cyl11
         C11SensorPositionFault : Bool;   // Cyl11
         C11SpareFault : Bool;
         C12GoWorkFault : Bool;   // Cyl12
         C12GoHomeFault : Bool;   // Cyl12
         C12SensorPositionFault : Bool;   // Cyl12
         C12SpareFault : Bool;
         C13GoWorkFault : Bool;   // Cyl13
         C13GoHomeFault : Bool;   // Cyl13
         C13SensorPositionFault : Bool;   // Cyl13
         C13SpareFault : Bool;
         C14GoWorkFault : Bool;   // Cyl14
         C14GoHomeFault : Bool;   // Cyl14
         C14SensorPositionFault : Bool;   // Cyl14
         C14SpareFault : Bool;
         C15GoWorkFault : Bool;   // Cyl15
         C15GoHomeFault : Bool;   // Cyl15
         C15SensorPositionFault : Bool;   // Cyl15
         C15SpareFault : Bool;
         C16GoWorkFault : Bool;   // Cyl16
         C16GoHomeFault : Bool;   // Cyl16
         C16SensorPositionFault : Bool;   // Cyl16
         C16SpareFault : Bool;
         C17GoWorkFault : Bool;   // Cyl17
         C17GoHomeFault : Bool;   // Cyl17
         C17SensorPositionFault : Bool;   // Cyl17
         C17SpareFault : Bool;
         C18GoWorkFault : Bool;   // Cyl18
         C18GoHomeFault : Bool;   // Cyl18
         C18SensorPositionFault : Bool;   // Cyl18
         C18SpareFault : Bool;
         C19GoWorkFault : Bool;   // Cyl19
         C19GoHomeFault : Bool;   // Cyl19
         C19SensorPositionFault : Bool;   // Cyl19
         C19SpareFault : Bool;
         C20GoWorkFault : Bool;   // Cyl20
         C20GoHomeFault : Bool;   // Cyl20
         C20SensorPositionFault : Bool;   // Cyl20
         C20SpareFault : Bool;
         C21GoWorkFault : Bool;   // Cyl21
         C21GoHomeFault : Bool;   // Cyl21
         C21SensorPositionFault : Bool;   // Cyl21
         C21SpareFault : Bool;
         C22GoWorkFault : Bool;   // Cyl22
         C22GoHomeFault : Bool;   // Cyl22
         C22SensorPositionFault : Bool;   // Cyl22
         C22SpareFault : Bool;
         C23GoWorkFault : Bool;   // Cyl23
         C23GoHomeFault : Bool;   // Cyl23
         C23SensorPositionFault : Bool;   // Cyl23
         C23SpareFault : Bool;
         C24GoWorkFault : Bool;   // Cyl24
         C24GoHomeFault : Bool;   // Cyl24
         C24SensorPositionFault : Bool;   // Cyl24
         C24SpareFault : Bool;
         C25GoWorkFault : Bool;   // Cyl25
         C25GoHomeFault : Bool;   // Cyl25
         C25SensorPositionFault : Bool;   // Cyl25
         C25SpareFault : Bool;
         C26GoWorkFault : Bool;   // Cyl26
         C26GoHomeFault : Bool;   // Cyl26
         C26SensorPositionFault : Bool;   // Cyl26
         C26SpareFault : Bool;
         C27GoWorkFault : Bool;   // Cyl27
         C27GoHomeFault : Bool;   // Cyl27
         C27SensorPositionFault : Bool;   // Cyl27
         C27SpareFault : Bool;
         C28GoWorkFault : Bool;   // Cyl28
         C28GoHomeFault : Bool;   // Cyl28
         C28SensorPositionFault : Bool;   // Cyl28
         C28SpareFault : Bool;
         C29GoWorkFault : Bool;   // Cyl29
         C29GoHomeFault : Bool;   // Cyl29
         C29SensorPositionFault : Bool;   // Cyl29
         C29SpareFault : Bool;
         C30GoWorkFault : Bool;   // Cyl30
         C30GoHomeFault : Bool;   // Cyl30
         C30SensorPositionFault : Bool;   // Cyl30
         C30SpareFault : Bool;
         C31GoWorkFault : Bool;   // Cyl31
         C31GoHomeFault : Bool;   // Cyl31
         C31SensorPositionFault : Bool;   // Cyl31
         C31SpareFault : Bool;
         C32GoWorkFault : Bool;   // Cyl32
         C32GoHomeFault : Bool;   // Cyl32
         C32SensorPositionFault : Bool;   // Cyl32
         C32SpareFault : Bool;
         C33GoWorkFault : Bool;   // Cyl33
         C33GoHomeFault : Bool;   // Cyl33
         C33SensorPositionFault : Bool;   // Cyl33
         C33SpareFault : Bool;
         C34GoWorkFault : Bool;   // Cyl34
         C34GoHomeFault : Bool;   // Cyl34
         C34SensorPositionFault : Bool;   // Cyl34
         C34SpareFault : Bool;
         C35GoWorkFault : Bool;   // Cyl35
         C35GoHomeFault : Bool;   // Cyl35
         C35SensorPositionFault : Bool;   // Cyl35
         C35SpareFault : Bool;
         C36GoWorkFault : Bool;   // Cyl36
         C36GoHomeFault : Bool;   // Cyl36
         C36SensorPositionFault : Bool;   // Cyl36
         C36SpareFault : Bool;
         C37GoWorkFault : Bool;   // Cyl37
         C37GoHomeFault : Bool;   // Cyl37
         C37SensorPositionFault : Bool;   // Cyl37
         C37SpareFault : Bool;
         C38GoWorkFault : Bool;   // Cyl38
         C38GoHomeFault : Bool;   // Cyl38
         C38SensorPositionFault : Bool;   // Cyl38
         C38SpareFault : Bool;
         C39GoWorkFault : Bool;   // Cyl39
         C39GoHomeFault : Bool;   // Cyl39
         C39SensorPositionFault : Bool;   // Cyl39
         C39SpareFault : Bool;
         C40GoWorkFault : Bool;   // Cyl40
         C40GoHomeFault : Bool;   // Cyl40
         C40SensorPositionFault : Bool;   // Cyl40
         C40SpareFault : Bool;
         C41GoWorkFault : Bool;   // Cyl41
         C41GoHomeFault : Bool;   // Cyl41
         C41SensorPositionFault : Bool;   // Cyl41
         C41SpareFault : Bool;
         C42GoWorkFault : Bool;   // Cyl42
         C42GoHomeFault : Bool;   // Cyl42
         C42SensorPositionFault : Bool;   // Cyl42
         C42SpareFault : Bool;
         C43GoWorkFault : Bool;   // Cyl43
         C43GoHomeFault : Bool;   // Cyl43
         C43SensorPositionFault : Bool;   // Cyl43
         C43SpareFault : Bool;
         C44GoWorkFault : Bool;   // Cyl44
         C44GoHomeFault : Bool;   // Cyl44
         C44SensorPositionFault : Bool;   // Cyl44
         C44SpareFault : Bool;
         C45GoWorkFault : Bool;   // Cyl45
         C45GoHomeFault : Bool;   // Cyl45
         C45SensorPositionFault : Bool;   // Cyl45
         C45SpareFault : Bool;
         C46GoWorkFault : Bool;   // Cyl46
         C46GoHomeFault : Bool;   // Cyl46
         C46SensorPositionFault : Bool;   // Cyl46
         C46SpareFault : Bool;
         C47GoWorkFault : Bool;   // Cyl47
         C47GoHomeFault : Bool;   // Cyl47
         C47SensorPositionFault : Bool;   // Cyl47
         C47SpareFault : Bool;
         C48GoWorkFault : Bool;   // Cyl48
         C48GoHomeFault : Bool;   // Cyl48
         C48SensorPositionFault : Bool;   // Cyl48
         C48SpareFault : Bool;
         C49GoWorkFault : Bool;   // Cyl49
         C49GoHomeFault : Bool;   // Cyl49
         C49SensorPositionFault : Bool;   // Cyl49
         C49SpareFault : Bool;
         C50GoWorkFault : Bool;   // Cyl50
         C50GoHomeFault : Bool;   // Cyl50
         C50SensorPositionFault : Bool;   // Cyl50
         C50SpareFault : Bool;
         C51GoWorkFault : Bool;   // Cyl51
         C51GoHomeFault : Bool;   // Cyl51
         C51SensorPositionFault : Bool;   // Cyl51
         C51SpareFault : Bool;
         C52GoWorkFault : Bool;   // Cyl52
         C52GoHomeFault : Bool;   // Cyl52
         C52SensorPositionFault : Bool;   // Cyl52
         C52SpareFault : Bool;
         C53GoWorkFault : Bool;   // Cyl53
         C53GoHomeFault : Bool;   // Cyl53
         C53SensorPositionFault : Bool;   // Cyl53
         C53SpareFault : Bool;
         C54GoWorkFault : Bool;   // Cyl54
         C54GoHomeFault : Bool;   // Cyl54
         C54SensorPositionFault : Bool;   // Cyl54
         C54SpareFault : Bool;
         C55GoWorkFault : Bool;   // Cyl55
         C55GoHomeFault : Bool;   // Cyl55
         C55SensorPositionFault : Bool;   // Cyl55
         C55SpareFault : Bool;
         C56GoWorkFault : Bool;   // Cyl56
         C56GoHomeFault : Bool;   // Cyl56
         C56SensorPositionFault : Bool;   // Cyl56
         C56SpareFault : Bool;
         C57GoWorkFault : Bool;   // Cyl57
         C57GoHomeFault : Bool;   // Cyl57
         C57SensorPositionFault : Bool;   // Cyl57
         C57SpareFault : Bool;
         C58GoWorkFault : Bool;   // Cyl58
         C58GoHomeFault : Bool;   // Cyl58
         C58SensorPositionFault : Bool;   // Cyl58
         C58SpareFault : Bool;
         C59GoWorkFault : Bool;   // Cyl59
         C59GoHomeFault : Bool;   // Cyl59
         C59SensorPositionFault : Bool;   // Cyl59
         C59SpareFault : Bool;
         C60GoWorkFault : Bool;   // Cyl60
         C60GoHomeFault : Bool;   // Cyl60
         C60SensorPositionFault : Bool;   // Cyl60
         C60SpareFault : Bool;
         C61GoWorkFault : Bool;   // Cyl61
         C61GoHomeFault : Bool;   // Cyl61
         C61SensorPositionFault : Bool;   // Cyl61
         C61SpareFault : Bool;
         C62GoWorkFault : Bool;   // Cyl62
         C62GoHomeFault : Bool;   // Cyl62
         C62SensorPositionFault : Bool;   // Cyl62
         C62SpareFault : Bool;
         C63GoWorkFault : Bool;   // Cyl63
         C63GoHomeFault : Bool;   // Cyl63
         C63SensorPositionFault : Bool;   // Cyl63
         C63SpareFault : Bool;
         C64GoWorkFault : Bool;   // Cyl64
         C64GoHomeFault : Bool;   // Cyl64
         C64SensorPositionFault : Bool;   // Cyl64
         C64SpareFault : Bool;
         C65GoWorkFault : Bool;   // Cyl65
         C65GoHomeFault : Bool;   // Cyl65
         C65SensorPositionFault : Bool;   // Cyl65
         C65SpareFault : Bool;
         C66GoWorkFault : Bool;   // Cyl66
         C66GoHomeFault : Bool;   // Cyl66
         C66SensorPositionFault : Bool;   // Cyl66
         C66SpareFault : Bool;
         C67GoWorkFault : Bool;   // Cyl67
         C67GoHomeFault : Bool;   // Cyl67
         C67SensorPositionFault : Bool;   // Cyl67
         C67SpareFault : Bool;
         C68GoWorkFault : Bool;   // Cyl68
         C68GoHomeFault : Bool;   // Cyl68
         C68SensorPositionFault : Bool;   // Cyl68
         C68SpareFault : Bool;
         C69GoWorkFault : Bool;   // Cyl69
         C69GoHomeFault : Bool;   // Cyl69
         C69SensorPositionFault : Bool;   // Cyl69
         C69SpareFault : Bool;
         C70GoWorkFault : Bool;   // Cyl70
         C70GoHomeFault : Bool;   // Cyl70
         C70SensorPositionFault : Bool;   // Cyl70
         C70SpareFault : Bool;
         C71GoWorkFault : Bool;   // Cyl71
         C71GoHomeFault : Bool;   // Cyl71
         C71SensorPositionFault : Bool;   // Cyl71
         C71SpareFault : Bool;
         C72GoWorkFault : Bool;   // Cyl72
         C72GoHomeFault : Bool;   // Cyl72
         C72SensorPositionFault : Bool;   // Cyl72
         C72SpareFault : Bool;
         C73GoWorkFault : Bool;   // Cyl73
         C73GoHomeFault : Bool;   // Cyl73
         C73SensorPositionFault : Bool;   // Cyl73
         C73SpareFault : Bool;
         C74GoWorkFault : Bool;   // Cyl74
         C74GoHomeFault : Bool;   // Cyl74
         C74SensorPositionFault : Bool;   // Cyl74
         C74SpareFault : Bool;
         C75GoWorkFault : Bool;   // Cyl75
         C75GoHomeFault : Bool;   // Cyl75
         C75SensorPositionFault : Bool;   // Cyl75
         C75SpareFault : Bool;
         C76GoWorkFault : Bool;   // Cyl76
         C76GoHomeFault : Bool;   // Cyl76
         C76SensorPositionFault : Bool;   // Cyl76
         C76SpareFault : Bool;
         C77GoWorkFault : Bool;   // Cyl77
         C77GoHomeFault : Bool;   // Cyl77
         C77SensorPositionFault : Bool;   // Cyl77
         C77SpareFault : Bool;
         C78GoWorkFault : Bool;   // Cyl78
         C78GoHomeFault : Bool;   // Cyl78
         C78SensorPositionFault : Bool;   // Cyl78
         C78SpareFault : Bool;
         C79GoWorkFault : Bool;   // Cyl79
         C79GoHomeFault : Bool;   // Cyl79
         C79SensorPositionFault : Bool;   // Cyl79
         C79SpareFault : Bool;
         C80GoWorkFault : Bool;   // Cyl80
         C80GoHomeFault : Bool;   // Cyl80
         C80SensorPositionFault : Bool;   // Cyl80
         C80SpareFault : Bool;
         C81GoWorkFault : Bool;   // Cyl81
         C81GoHomeFault : Bool;   // Cyl81
         C81SensorPositionFault : Bool;   // Cyl81
         C81SpareFault : Bool;
         C82GoWorkFault : Bool;   // Cyl82
         C82GoHomeFault : Bool;   // Cyl82
         C82SensorPositionFault : Bool;   // Cyl82
         C82SpareFault : Bool;
         C83GoWorkFault : Bool;   // Cyl83
         C83GoHomeFault : Bool;   // Cyl83
         C83SensorPositionFault : Bool;   // Cyl83
         C83SpareFault : Bool;
         C84GoWorkFault : Bool;   // Cyl84
         C84GoHomeFault : Bool;   // Cyl84
         C84SensorPositionFault : Bool;   // Cyl84
         C84SpareFault : Bool;
         C85GoWorkFault : Bool;   // Cyl85
         C85GoHomeFault : Bool;   // Cyl85
         C85SensorPositionFault : Bool;   // Cyl85
         C85SpareFault : Bool;
         C86GoWorkFault : Bool;   // Cyl86
         C86GoHomeFault : Bool;   // Cyl86
         C86SensorPositionFault : Bool;   // Cyl86
         C86SpareFault : Bool;
         C87GoWorkFault : Bool;   // Cyl87
         C87GoHomeFault : Bool;   // Cyl87
         C87SensorPositionFault : Bool;   // Cyl87
         C87SpareFault : Bool;
         C88GoWorkFault : Bool;   // Cyl88
         C88GoHomeFault : Bool;   // Cyl88
         C88SensorPositionFault : Bool;   // Cyl88
         C88SpareFault : Bool;
         C89GoWorkFault : Bool;   // Cyl89
         C89GoHomeFault : Bool;   // Cyl89
         C89SensorPositionFault : Bool;   // Cyl89
         C89SpareFault : Bool;
         C90GoWorkFault : Bool;   // Cyl90
         C90GoHomeFault : Bool;   // Cyl90
         C90SensorPositionFault : Bool;   // Cyl90
         C90SpareFault : Bool;
         C91GoWorkFault : Bool;   // Cyl91
         C91GoHomeFault : Bool;   // Cyl91
         C91SensorPositionFault : Bool;   // Cyl91
         C91SpareFault : Bool;
         C92GoWorkFault : Bool;   // Cyl92
         C92GoHomeFault : Bool;   // Cyl92
         C92SensorPositionFault : Bool;   // Cyl92
         C92SpareFault : Bool;
         C93GoWorkFault : Bool;   // Cyl93
         C93GoHomeFault : Bool;   // Cyl93
         C93SensorPositionFault : Bool;   // Cyl93
         C93SpareFault : Bool;
         C94GoWorkFault : Bool;   // Cyl94
         C94GoHomeFault : Bool;   // Cyl94
         C94SensorPositionFault : Bool;   // Cyl94
         C94SpareFault : Bool;
         C95GoWorkFault : Bool;   // Cyl95
         C95GoHomeFault : Bool;   // Cyl95
         C95SensorPositionFault : Bool;   // Cyl95
         C95SpareFault : Bool;
         C96GoWorkFault : Bool;   // Cyl96
         C96GoHomeFault : Bool;   // Cyl96
         C96SensorPositionFault : Bool;   // Cyl96
         C96SpareFault : Bool;
         C97GoWorkFault : Bool;   // Cyl97
         C97GoHomeFault : Bool;   // Cyl97
         C97SensorPositionFault : Bool;   // Cyl97
         C97SpareFault : Bool;
         C98GoWorkFault : Bool;   // Cyl98
         C98GoHomeFault : Bool;   // Cyl98
         C98SensorPositionFault : Bool;   // Cyl98
         C98SpareFault : Bool;
         C99GoWorkFault : Bool;   // Cyl99
         C99GoHomeFault : Bool;   // Cyl99
         C99SensorPositionFault : Bool;   // Cyl99
         C99SpareFault : Bool;
         C100GoWorkFault : Bool;   // Cyl100
         C100GoHomeFault : Bool;   // Cyl100
         C100SensorPositionFault : Bool;   // Cyl100
         C100SpareFault : Bool;
         C101GoWorkFault : Bool;   // Cyl101
         C101GoHomeFault : Bool;   // Cyl101
         C101SensorPositionFault : Bool;   // Cyl101
         C101SpareFault : Bool;
         C102GoWorkFault : Bool;   // Cyl102
         C102GoHomeFault : Bool;   // Cyl102
         C102SensorPositionFault : Bool;   // Cyl102
         C102SpareFault : Bool;
         C103GoWorkFault : Bool;   // Cyl103
         C103GoHomeFault : Bool;   // Cyl103
         C103SensorPositionFault : Bool;   // Cyl103
         C103SpareFault : Bool;
         C104GoWorkFault : Bool;   // Cyl104
         C104GoHomeFault : Bool;   // Cyl104
         C104SensorPositionFault : Bool;   // Cyl104
         C104SpareFault : Bool;
         C105GoWorkFault : Bool;   // Cyl105
         C105GoHomeFault : Bool;   // Cyl105
         C105SensorPositionFault : Bool;   // Cyl105
         C105SpareFault : Bool;
         C106GoWorkFault : Bool;   // Cyl106
         C106GoHomeFault : Bool;   // Cyl106
         C106SensorPositionFault : Bool;   // Cyl106
         C106SpareFault : Bool;
         C107GoWorkFault : Bool;   // Cyl107
         C107GoHomeFault : Bool;   // Cyl107
         C107SensorPositionFault : Bool;   // Cyl107
         C107SpareFault : Bool;
         C108GoWorkFault : Bool;   // Cyl108
         C108GoHomeFault : Bool;   // Cyl108
         C108SensorPositionFault : Bool;   // Cyl108
         C108SpareFault : Bool;
         C109GoWorkFault : Bool;   // Cyl109
         C109GoHomeFault : Bool;   // Cyl109
         C109SensorPositionFault : Bool;   // Cyl109
         C109SpareFault : Bool;
         C110GoWorkFault : Bool;   // Cyl110
         C110GoHomeFault : Bool;   // Cyl110
         C110SensorPositionFault : Bool;   // Cyl110
         C110SpareFault : Bool;
         C111GoWorkFault : Bool;   // Cyl111
         C111GoHomeFault : Bool;   // Cyl111
         C111SensorPositionFault : Bool;   // Cyl111
         C111SpareFault : Bool;
         C112GoWorkFault : Bool;   // Cyl112
         C112GoHomeFault : Bool;   // Cyl112
         C112SensorPositionFault : Bool;   // Cyl112
         C112SpareFault : Bool;
         C113GoWorkFault : Bool;   // Cyl113
         C113GoHomeFault : Bool;   // Cyl113
         C113SensorPositionFault : Bool;   // Cyl113
         C113SpareFault : Bool;
         C114GoWorkFault : Bool;   // Cyl114
         C114GoHomeFault : Bool;   // Cyl114
         C114SensorPositionFault : Bool;   // Cyl114
         C114SpareFault : Bool;
         C115GoWorkFault : Bool;   // Cyl115
         C115GoHomeFault : Bool;   // Cyl115
         C115SensorPositionFault : Bool;   // Cyl115
         C115SpareFault : Bool;
         C116GoWorkFault : Bool;   // Cyl116
         C116GoHomeFault : Bool;   // Cyl116
         C116SensorPositionFault : Bool;   // Cyl116
         C116SpareFault : Bool;
         C117GoWorkFault : Bool;   // Cyl117
         C117GoHomeFault : Bool;   // Cyl117
         C117SensorPositionFault : Bool;   // Cyl117
         C117SpareFault : Bool;
         C118GoWorkFault : Bool;   // Cyl118
         C118GoHomeFault : Bool;   // Cyl118
         C118SensorPositionFault : Bool;   // Cyl118
         C118SpareFault : Bool;
         C119GoWorkFault : Bool;   // Cyl119
         C119GoHomeFault : Bool;   // Cyl119
         C119SensorPositionFault : Bool;   // Cyl119
         C119SpareFault : Bool;
         C120GoWorkFault : Bool;   // Cyl120
         C120GoHomeFault : Bool;   // Cyl120
         C120SensorPositionFault : Bool;   // Cyl120
         C120SpareFault : Bool;
         C121GoWorkFault : Bool;   // Cyl121
         C121GoHomeFault : Bool;   // Cyl121
         C121SensorPositionFault : Bool;   // Cyl121
         C121SpareFault : Bool;
         C122GoWorkFault : Bool;   // Cyl122
         C122GoHomeFault : Bool;   // Cyl122
         C122SensorPositionFault : Bool;   // Cyl122
         C122SpareFault : Bool;
         C123GoWorkFault : Bool;   // Cyl123
         C123GoHomeFault : Bool;   // Cyl123
         C123SensorPositionFault : Bool;   // Cyl123
         C123SpareFault : Bool;
         C124GoWorkFault : Bool;   // Cyl124
         C124GoHomeFault : Bool;   // Cyl124
         C124SensorPositionFault : Bool;   // Cyl124
         C124SpareFault : Bool;
         C125GoWorkFault : Bool;   // Cyl125
         C125GoHomeFault : Bool;   // Cyl125
         C125SensorPositionFault : Bool;   // Cyl125
         C125SpareFault : Bool;
         C126GoWorkFault : Bool;   // Cyl126
         C126GoHomeFault : Bool;   // Cyl126
         C126SensorPositionFault : Bool;   // Cyl126
         C126SpareFault : Bool;
         C127GoWorkFault : Bool;   // Cyl127
         C127GoHomeFault : Bool;   // Cyl127
         C127SensorPositionFault : Bool;   // Cyl127
         C127SpareFault : Bool;
         C128GoWorkFault : Bool;   // Cyl128
         C128GoHomeFault : Bool;   // Cyl128
         C128SensorPositionFault : Bool;   // Cyl128
         C128SpareFault : Bool;
         C129GoWorkFault : Bool;   // Cyl129
         C129GoHomeFault : Bool;   // Cyl129
         C129SensorPositionFault : Bool;   // Cyl129
         C129SpareFault : Bool;
         C130GoWorkFault : Bool;   // Cyl130
         C130GoHomeFault : Bool;   // Cyl130
         C130SensorPositionFault : Bool;   // Cyl130
         C130SpareFault : Bool;
         C131GoWorkFault : Bool;   // Cyl131
         C131GoHomeFault : Bool;   // Cyl131
         C131SensorPositionFault : Bool;   // Cyl131
         C131SpareFault : Bool;
         C132GoWorkFault : Bool;   // Cyl132
         C132GoHomeFault : Bool;   // Cyl132
         C132SensorPositionFault : Bool;   // Cyl132
         C132SpareFault : Bool;
         C133GoWorkFault : Bool;   // Cyl133
         C133GoHomeFault : Bool;   // Cyl133
         C133SensorPositionFault : Bool;   // Cyl133
         C133SpareFault : Bool;
         C134GoWorkFault : Bool;   // Cyl134
         C134GoHomeFault : Bool;   // Cyl134
         C134SensorPositionFault : Bool;   // Cyl134
         C134SpareFault : Bool;
         C135GoWorkFault : Bool;   // Cyl135
         C135GoHomeFault : Bool;   // Cyl135
         C135SensorPositionFault : Bool;   // Cyl135
         C135SpareFault : Bool;
         C136GoWorkFault : Bool;   // Cyl136
         C136GoHomeFault : Bool;   // Cyl136
         C136SensorPositionFault : Bool;   // Cyl136
         C136SpareFault : Bool;
         C137GoWorkFault : Bool;   // Cyl137
         C137GoHomeFault : Bool;   // Cyl137
         C137SensorPositionFault : Bool;   // Cyl137
         C137SpareFault : Bool;
         C138GoWorkFault : Bool;   // Cyl138
         C138GoHomeFault : Bool;   // Cyl138
         C138SensorPositionFault : Bool;   // Cyl138
         C138SpareFault : Bool;
         C139GoWorkFault : Bool;   // Cyl139
         C139GoHomeFault : Bool;   // Cyl139
         C139SensorPositionFault : Bool;   // Cyl139
         C139SpareFault : Bool;
         C140GoWorkFault : Bool;   // Cyl140
         C140GoHomeFault : Bool;   // Cyl140
         C140SensorPositionFault : Bool;   // Cyl140
         C140SpareFault : Bool;
         C141GoWorkFault : Bool;   // Cyl141
         C141GoHomeFault : Bool;   // Cyl141
         C141SensorPositionFault : Bool;   // Cyl141
         C141SpareFault : Bool;
         C142GoWorkFault : Bool;   // Cyl142
         C142GoHomeFault : Bool;   // Cyl142
         C142SensorPositionFault : Bool;   // Cyl142
         C142SpareFault : Bool;
         C143GoWorkFault : Bool;   // Cyl143
         C143GoHomeFault : Bool;   // Cyl143
         C143SensorPositionFault : Bool;   // Cyl143
         C143SpareFault : Bool;
         C144GoWorkFault : Bool;   // Cyl144
         C144GoHomeFault : Bool;   // Cyl144
         C144SensorPositionFault : Bool;   // Cyl144
         C144SpareFault : Bool;
         C145GoWorkFault : Bool;   // Cyl145
         C145GoHomeFault : Bool;   // Cyl145
         C145SensorPositionFault : Bool;   // Cyl145
         C145SpareFault : Bool;
         C146GoWorkFault : Bool;   // Cyl146
         C146GoHomeFault : Bool;   // Cyl146
         C146SensorPositionFault : Bool;   // Cyl146
         C146SpareFault : Bool;
         C147GoWorkFault : Bool;   // Cyl147
         C147GoHomeFault : Bool;   // Cyl147
         C147SensorPositionFault : Bool;   // Cyl147
         C147SpareFault : Bool;
         C148GoWorkFault : Bool;   // Cyl148
         C148GoHomeFault : Bool;   // Cyl148
         C148SensorPositionFault : Bool;   // Cyl148
         C148SpareFault : Bool;
         C149GoWorkFault : Bool;   // Cyl149
         C149GoHomeFault : Bool;   // Cyl149
         C149SensorPositionFault : Bool;   // Cyl149
         C149SpareFault : Bool;
         C150GoWorkFault : Bool;   // Cyl150
         C150GoHomeFault : Bool;   // Cyl150
         C150SensorPositionFault : Bool;   // Cyl150
         C150SpareFault : Bool;
         C151GoWorkFault : Bool;   // Cyl151
         C151GoHomeFault : Bool;   // Cyl151
         C151SensorPositionFault : Bool;   // Cyl151
         C151SpareFault : Bool;
         C152GoWorkFault : Bool;   // Cyl152
         C152GoHomeFault : Bool;   // Cyl152
         C152SensorPositionFault : Bool;   // Cyl152
         C152SpareFault : Bool;
         C153GoWorkFault : Bool;   // Cyl153
         C153GoHomeFault : Bool;   // Cyl153
         C153SensorPositionFault : Bool;   // Cyl153
         C153SpareFault : Bool;
         C154GoWorkFault : Bool;   // Cyl154
         C154GoHomeFault : Bool;   // Cyl154
         C154SensorPositionFault : Bool;   // Cyl154
         C154SpareFault : Bool;
         C155GoWorkFault : Bool;   // Cyl155
         C155GoHomeFault : Bool;   // Cyl155
         C155SensorPositionFault : Bool;   // Cyl155
         C155SpareFault : Bool;
         C156GoWorkFault : Bool;   // Cyl156
         C156GoHomeFault : Bool;   // Cyl156
         C156SensorPositionFault : Bool;   // Cyl156
         C156SpareFault : Bool;
         C157GoWorkFault : Bool;   // Cyl157
         C157GoHomeFault : Bool;   // Cyl157
         C157SensorPositionFault : Bool;   // Cyl157
         C157SpareFault : Bool;
         C158GoWorkFault : Bool;   // Cyl158
         C158GoHomeFault : Bool;   // Cyl158
         C158SensorPositionFault : Bool;   // Cyl158
         C158SpareFault : Bool;
         C159GoWorkFault : Bool;   // Cyl159
         C159GoHomeFault : Bool;   // Cyl159
         C159SensorPositionFault : Bool;   // Cyl159
         C159SpareFault : Bool;
         C160GoWorkFault : Bool;   // Cyl160
         C160GoHomeFault : Bool;   // Cyl160
         C160SensorPositionFault : Bool;   // Cyl160
         C160SpareFault : Bool;
         C161GoWorkFault : Bool;   // Cyl161
         C161GoHomeFault : Bool;   // Cyl161
         C161SensorPositionFault : Bool;   // Cyl161
         C161SpareFault : Bool;
         C162GoWorkFault : Bool;   // Cyl162
         C162GoHomeFault : Bool;   // Cyl162
         C162SensorPositionFault : Bool;   // Cyl162
         C162SpareFault : Bool;
         C163GoWorkFault : Bool;   // Cyl163
         C163GoHomeFault : Bool;   // Cyl163
         C163SensorPositionFault : Bool;   // Cyl163
         C163SpareFault : Bool;
         C164GoWorkFault : Bool;   // Cyl164
         C164GoHomeFault : Bool;   // Cyl164
         C164SensorPositionFault : Bool;   // Cyl164
         C164SpareFault : Bool;
         C165GoWorkFault : Bool;   // Cyl165
         C165GoHomeFault : Bool;   // Cyl165
         C165SensorPositionFault : Bool;   // Cyl165
         C165SpareFault : Bool;
         C166GoWorkFault : Bool;   // Cyl166
         C166GoHomeFault : Bool;   // Cyl166
         C166SensorPositionFault : Bool;   // Cyl166
         C166SpareFault : Bool;
         C167GoWorkFault : Bool;   // Cyl167
         C167GoHomeFault : Bool;   // Cyl167
         C167SensorPositionFault : Bool;   // Cyl167
         C167SpareFault : Bool;
         C168GoWorkFault : Bool;   // Cyl168
         C168GoHomeFault : Bool;   // Cyl168
         C168SensorPositionFault : Bool;   // Cyl168
         C168SpareFault : Bool;
         C169GoWorkFault : Bool;   // Cyl169
         C169GoHomeFault : Bool;   // Cyl169
         C169SensorPositionFault : Bool;   // Cyl169
         C169SpareFault : Bool;
         C170GoWorkFault : Bool;   // Cyl170
         C170GoHomeFault : Bool;   // Cyl170
         C170SensorPositionFault : Bool;   // Cyl170
         C170SpareFault : Bool;
         C171GoWorkFault : Bool;   // Cyl171
         C171GoHomeFault : Bool;   // Cyl171
         C171SensorPositionFault : Bool;   // Cyl171
         C171SpareFault : Bool;
         C172GoWorkFault : Bool;   // Cyl172
         C172GoHomeFault : Bool;   // Cyl172
         C172SensorPositionFault : Bool;   // Cyl172
         C172SpareFault : Bool;
         C173GoWorkFault : Bool;   // Cyl173
         C173GoHomeFault : Bool;   // Cyl173
         C173SensorPositionFault : Bool;   // Cyl173
         C173SpareFault : Bool;
         C174GoWorkFault : Bool;   // Cyl174
         C174GoHomeFault : Bool;   // Cyl174
         C174SensorPositionFault : Bool;   // Cyl174
         C174SpareFault : Bool;
         C175GoWorkFault : Bool;   // Cyl175
         C175GoHomeFault : Bool;   // Cyl175
         C175SensorPositionFault : Bool;   // Cyl175
         C175SpareFault : Bool;
         C176GoWorkFault : Bool;   // Cyl176
         C176GoHomeFault : Bool;   // Cyl176
         C176SensorPositionFault : Bool;   // Cyl176
         C176SpareFault : Bool;
         C177GoWorkFault : Bool;   // Cyl177
         C177GoHomeFault : Bool;   // Cyl177
         C177SensorPositionFault : Bool;   // Cyl177
         C177SpareFault : Bool;
         C178GoWorkFault : Bool;   // Cyl178
         C178GoHomeFault : Bool;   // Cyl178
         C178SensorPositionFault : Bool;   // Cyl178
         C178SpareFault : Bool;
         C179GoWorkFault : Bool;   // Cyl179
         C179GoHomeFault : Bool;   // Cyl179
         C179SensorPositionFault : Bool;   // Cyl179
         C179SpareFault : Bool;
         C180GoWorkFault : Bool;   // Cyl180
         C180GoHomeFault : Bool;   // Cyl180
         C180SensorPositionFault : Bool;   // Cyl180
         C180SpareFault : Bool;
         C181GoWorkFault : Bool;   // Cyl181
         C181GoHomeFault : Bool;   // Cyl181
         C181SensorPositionFault : Bool;   // Cyl181
         C181SpareFault : Bool;
         C182GoWorkFault : Bool;   // Cyl182
         C182GoHomeFault : Bool;   // Cyl182
         C182SensorPositionFault : Bool;   // Cyl182
         C182SpareFault : Bool;
         C183GoWorkFault : Bool;   // Cyl183
         C183GoHomeFault : Bool;   // Cyl183
         C183SensorPositionFault : Bool;   // Cyl183
         C183SpareFault : Bool;
         C184GoWorkFault : Bool;   // Cyl184
         C184GoHomeFault : Bool;   // Cyl184
         C184SensorPositionFault : Bool;   // Cyl184
         C184SpareFault : Bool;
         C185GoWorkFault : Bool;   // Cyl185
         C185GoHomeFault : Bool;   // Cyl185
         C185SensorPositionFault : Bool;   // Cyl185
         C185SpareFault : Bool;
         C186GoWorkFault : Bool;   // Cyl186
         C186GoHomeFault : Bool;   // Cyl186
         C186SensorPositionFault : Bool;   // Cyl186
         C186SpareFault : Bool;
         C187GoWorkFault : Bool;   // Cyl187
         C187GoHomeFault : Bool;   // Cyl187
         C187SensorPositionFault : Bool;   // Cyl187
         C187SpareFault : Bool;
         C188GoWorkFault : Bool;   // Cyl188
         C188GoHomeFault : Bool;   // Cyl188
         C188SensorPositionFault : Bool;   // Cyl188
         C188SpareFault : Bool;
         C189GoWorkFault : Bool;   // Cyl189
         C189GoHomeFault : Bool;   // Cyl189
         C189SensorPositionFault : Bool;   // Cyl189
         C189SpareFault : Bool;
         C190GoWorkFault : Bool;   // Cyl190
         C190GoHomeFault : Bool;   // Cyl190
         C190SensorPositionFault : Bool;   // Cyl190
         C190SpareFault : Bool;
         C191GoWorkFault : Bool;   // Cyl191
         C191GoHomeFault : Bool;   // Cyl191
         C191SensorPositionFault : Bool;   // Cyl191
         C191SpareFault : Bool;
         C192GoWorkFault : Bool;   // Cyl192
         C192GoHomeFault : Bool;   // Cyl192
         C192SensorPositionFault : Bool;   // Cyl192
         C192SpareFault : Bool;
         C193GoWorkFault : Bool;   // Cyl193
         C193GoHomeFault : Bool;   // Cyl193
         C193SensorPositionFault : Bool;   // Cyl193
         C193SpareFault : Bool;
         C194GoWorkFault : Bool;   // Cyl194
         C194GoHomeFault : Bool;   // Cyl194
         C194SensorPositionFault : Bool;   // Cyl194
         C194SpareFault : Bool;
         C195GoWorkFault : Bool;   // Cyl195
         C195GoHomeFault : Bool;   // Cyl195
         C195SensorPositionFault : Bool;   // Cyl195
         C195SpareFault : Bool;
         C196GoWorkFault : Bool;   // Cyl196
         C196GoHomeFault : Bool;   // Cyl196
         C196SensorPositionFault : Bool;   // Cyl196
         C196SpareFault : Bool;
         C197GoWorkFault : Bool;   // Cyl197
         C197GoHomeFault : Bool;   // Cyl197
         C197SensorPositionFault : Bool;   // Cyl197
         C197SpareFault : Bool;
         C198GoWorkFault : Bool;   // Cyl198
         C198GoHomeFault : Bool;   // Cyl198
         C198SensorPositionFault : Bool;   // Cyl198
         C198SpareFault : Bool;
         C199GoWorkFault : Bool;   // Cyl199
         C199GoHomeFault : Bool;   // Cyl199
         C199SensorPositionFault : Bool;   // Cyl199
         C199SpareFault : Bool;
         C200GoWorkFault : Bool;   // Cyl200
         C200GoHomeFault : Bool;   // Cyl200
         C200SensorPositionFault : Bool;   // Cyl200
         C200SpareFault : Bool;
      END_STRUCT;
      "A" : Struct   // D-提升机顶升入口电机1错误
         A1TableScan : Struct   // Conveyor motor Breaker tripped,please check input Ix.x
            LightCuritTouch : Bool;
            ScanCodeNG : Bool;
            "3" : Bool;
            "4" : Bool;
            "5" : Bool;
            "6" : Bool;
            "7" : Bool;
            "8" : Bool;
            "9" : Bool;
            "10" : Bool;
            "11" : Bool;
            "12" : Bool;
            "13" : Bool;
            "14" : Bool;
            "15" : Bool;
            "16" : Bool;
         END_STRUCT;
         A1TableUnloading : Struct   // Conveyor motor start abnormal,please check output Qx.x
            LackMaterial : Bool;
            RingCheckExist : Bool;
            "3" : Bool;
            "4" : Bool;
            "5" : Bool;
            "6" : Bool;
            "7" : Bool;
            "8" : Bool;
            "9" : Bool;
            "10" : Bool;
            "11" : Bool;
            "12" : Bool;
            "13" : Bool;
            "14" : Bool;
            "15" : Bool;
            "16" : Bool;
         END_STRUCT;
         A1RotaryScan : Struct
            ProductAnomaly : Bool;
            PartMissing : Bool;
            "3" : Bool;
            "4" : Bool;
            "5" : Bool;
            "6" : Bool;
            "7" : Bool;
            "8" : Bool;
            "9" : Bool;
            "10" : Bool;
            "11" : Bool;
            "12" : Bool;
            "13" : Bool;
            "14" : Bool;
            "15" : Bool;
            "16" : Bool;
         END_STRUCT;
         A1FixtureCodeScan : Struct
            ReadNG_1 : Bool;
            ReadNG_2 : Bool;
            ReadNG_3 : Bool;
            ReadNG_4 : Bool;
            ReadNG_5 : Bool;
            ReadNG_6 : Bool;
            ReadNG_7 : Bool;
            ReadNG_8 : Bool;
            ReadNG_9 : Bool;
            ReadNG_10 : Bool;
            ReadNG_11 : Bool;
            ReadNG_12 : Bool;
            ReadNG_13 : Bool;
            "14" : Bool;
            "15" : Bool;
            "16" : Bool;
         END_STRUCT;
         A2TableScan : Struct
            LightCuritTouch : Bool;
            ScanCodeNG : Bool;
            "3" : Bool;
            "4" : Bool;
            "5" : Bool;
            "6" : Bool;
            "7" : Bool;
            "8" : Bool;
            "9" : Bool;
            "10" : Bool;
            "11" : Bool;
            "12" : Bool;
            "13" : Bool;
            "14" : Bool;
            "15" : Bool;
            "16" : Bool;
         END_STRUCT;
         A2TableUnloading : Struct
            LackMaterial : Bool;
            RingCheckExist : Bool;
            "3" : Bool;
            "4" : Bool;
            "5" : Bool;
            "6" : Bool;
            "7" : Bool;
            "8" : Bool;
            "9" : Bool;
            "10" : Bool;
            "11" : Bool;
            "12" : Bool;
            "13" : Bool;
            "14" : Bool;
            "15" : Bool;
            "16" : Bool;
         END_STRUCT;
         A2RotaryScan : Struct
            "1" : Bool;
            "2" : Bool;
            "3" : Bool;
            "4" : Bool;
            "5" : Bool;
            "6" : Bool;
            "7" : Bool;
            "8" : Bool;
            "9" : Bool;
            "10" : Bool;
            "11" : Bool;
            "12" : Bool;
            "13" : Bool;
            "14" : Bool;
            "15" : Bool;
            "16" : Bool;
         END_STRUCT;
         A2FixtureCodeScan : Struct
            ReadNG_1 : Bool;
            ReadNG_2 : Bool;
            ReadNG_3 : Bool;
            ReadNG_4 : Bool;
            ReadNG_5 : Bool;
            ReadNG_6 : Bool;
            ReadNG_7 : Bool;
            ReadNG_8 : Bool;
            ReadNG_9 : Bool;
            ReadNG_10 : Bool;
            ReadNG_11 : Bool;
            ReadNG_12 : Bool;
            ReadNG_13 : Bool;
            "14" : Bool;
            "15" : Bool;
            "16" : Bool;
         END_STRUCT;
         Other : Struct
            Servo_380A1 : Bool;
            Servo_381A1 : Bool;
            Servo_383A1 : Bool;
            "4" : Bool;
            "5" : Bool;
            "6" : Bool;
            "7" : Bool;
            "8" : Bool;
            "9" : Bool;
            "10" : Bool;
            "11" : Bool;
            "12" : Bool;
            "13" : Bool;
            "14" : Bool;
            "15" : Bool;
            "16" : Bool;
         END_STRUCT;
         A_Spare_2 : Struct
            Servo_380A1 : Bool;
            Servo_381A1 : Bool;
            Scan_800A1 : Bool;
            Scan_801A1 : Bool;
            Scan_804A1 : Bool;
            "6" : Bool;
            "7" : Bool;
            "8" : Bool;
            "9" : Bool;
            "10" : Bool;
            "11" : Bool;
            "12" : Bool;
            "13" : Bool;
            "14" : Bool;
            "15" : Bool;
            "16" : Bool;
         END_STRUCT;
      END_STRUCT;
      "B" : Struct   // D-提升机顶升出口电机1错误
         B1Press : Struct   // Conveyor motor Breaker tripped,please check input Ix.x
            StatusError : Bool;
            ShaftSensorCheckError : Bool;
            RingSensorCheckError : Bool;
            "4" : Bool;
            "5" : Bool;
            "6" : Bool;
            "7" : Bool;
            "8" : Bool;
            "9" : Bool;
            "10" : Bool;
            "11" : Bool;
            "12" : Bool;
            "13" : Bool;
            "14" : Bool;
            "15" : Bool;
            "16" : Bool;
         END_STRUCT;
         B2Press : Struct   // Conveyor motor start abnormal,please check output Qx.x
            StatusError : Bool;
            ShaftSensorCheckError : Bool;
            RingSensorCheckError : Bool;
            "4" : Bool;
            "5" : Bool;
            "6" : Bool;
            "7" : Bool;
            "8" : Bool;
            "9" : Bool;
            "10" : Bool;
            "11" : Bool;
            "12" : Bool;
            "13" : Bool;
            "14" : Bool;
            "15" : Bool;
            "16" : Bool;
         END_STRUCT;
         B_Spare_1 : Struct
            Kistler_Press1_372A1 : Bool;
            Scan_806A1 : Bool;
            Kistler_Press2_375A1 : Bool;
            "4" : Bool;
            "5" : Bool;
            "6" : Bool;
            "7" : Bool;
            "8" : Bool;
            "9" : Bool;
            "10" : Bool;
            "11" : Bool;
            "12" : Bool;
            "13" : Bool;
            "14" : Bool;
            "15" : Bool;
            "16" : Bool;
         END_STRUCT;
         B_Spare_2 : Struct
            "1" : Bool;
            "2" : Bool;
            "3" : Bool;
            "4" : Bool;
            "5" : Bool;
            "6" : Bool;
            "7" : Bool;
            "8" : Bool;
            "9" : Bool;
            "10" : Bool;
            "11" : Bool;
            "12" : Bool;
            "13" : Bool;
            "14" : Bool;
            "15" : Bool;
            "16" : Bool;
         END_STRUCT;
         B_Spare_3 : Struct
            "1" : Bool;
            "2" : Bool;
            "3" : Bool;
            "4" : Bool;
            "5" : Bool;
            "6" : Bool;
            "7" : Bool;
            "8" : Bool;
            "9" : Bool;
            "10" : Bool;
            "11" : Bool;
            "12" : Bool;
            "13" : Bool;
            "14" : Bool;
            "15" : Bool;
            "16" : Bool;
         END_STRUCT;
      END_STRUCT;
      C : Struct   // E-线体线体电机1错误
         CGlueing : Struct   // Conveyor motor Breaker tripped,please check input Ix.x
            SysError : Bool;
            StatusError : Bool;
            Servo_383A1 : Bool;
            Z : Bool;
            X : Bool;
            Y : Bool;
            "7" : Bool;
            "8" : Bool;
            "9" : Bool;
            "10" : Bool;
            "11" : Bool;
            "12" : Bool;
            "13" : Bool;
            "14" : Bool;
            "15" : Bool;
            "16" : Bool;
         END_STRUCT;
         Other : Struct
            Servo_383A1 : Bool;
            Z : Bool;
            X : Bool;
            Y : Bool;
            "5" : Bool;
            "6" : Bool;
            "7" : Bool;
            "8" : Bool;
            "9" : Bool;
            "10" : Bool;
            "11" : Bool;
            "12" : Bool;
            "13" : Bool;
            "14" : Bool;
            "15" : Bool;
            "16" : Bool;
         END_STRUCT;
         C_Spare_2 : Struct
            Servo_382A1 : Bool;
            IV3_810A1 : Bool;
            IV3_811A1 : Bool;
            GluingDeviceReady : Bool;
            GluingFault : Bool;
            GluingRefillTank : Bool;
            GluingTankEmpty : Bool;
            "8" : Bool;
            "9" : Bool;
            "10" : Bool;
            "11" : Bool;
            "12" : Bool;
            "13" : Bool;
            "14" : Bool;
            "15" : Bool;
            "16" : Bool;
         END_STRUCT;
         C_Spare_3 : Struct
            "1" : Bool;
            "2" : Bool;
            "3" : Bool;
            "4" : Bool;
            "5" : Bool;
            "6" : Bool;
            "7" : Bool;
            "8" : Bool;
            "9" : Bool;
            "10" : Bool;
            "11" : Bool;
            "12" : Bool;
            "13" : Bool;
            "14" : Bool;
            "15" : Bool;
            "16" : Bool;
         END_STRUCT;
         C_Spare_4 : Struct
            "1" : Bool;
            "2" : Bool;
            "3" : Bool;
            "4" : Bool;
            "5" : Bool;
            "6" : Bool;
            "7" : Bool;
            "8" : Bool;
            "9" : Bool;
            "10" : Bool;
            "11" : Bool;
            "12" : Bool;
            "13" : Bool;
            "14" : Bool;
            "15" : Bool;
            "16" : Bool;
         END_STRUCT;
      END_STRUCT;
      "E" : Struct   // 上料扫码错误
         NG_1 : Struct
            ShaftScanNGFull : Bool;
            PressNGFull : Bool;
            RingScanNGFull : Bool;
            ShaftScanStatus : Bool;
            PressNGStatus : Bool;
            RingScanNGStatus : Bool;
            "NG 1 DoorOpen" : Bool;
            "NG 2 DoorOpen" : Bool;
            "9" : Bool;
            "10" : Bool;
            "11" : Bool;
            "12" : Bool;
            "13" : Bool;
            "14" : Bool;
            "15" : Bool;
            "16" : Bool;
         END_STRUCT;
         NG_2 : Struct
            "Press/GlueNGFull" : Bool;
            MagnetNGFull : Bool;
            RingScanNGFull : Bool;
            "Press/GlueNGStatus" : Bool;
            MagnetNGStatus : Bool;
            RingScanNGStatus : Bool;
            "7" : Bool;
            "8" : Bool;
            "9" : Bool;
            "10" : Bool;
            "11" : Bool;
            "12" : Bool;
            "13" : Bool;
            "14" : Bool;
            "15" : Bool;
            "16" : Bool;
         END_STRUCT;
         E_Spare_1 : Struct
            "1" : Bool;
            "2" : Bool;
            "3" : Bool;
            "4" : Bool;
            "5" : Bool;
            "6" : Bool;
            "7" : Bool;
            "8" : Bool;
            "9" : Bool;
            "10" : Bool;
            "11" : Bool;
            "12" : Bool;
            "13" : Bool;
            "14" : Bool;
            "15" : Bool;
            "16" : Bool;
         END_STRUCT;
         E_Spare_2 : Struct
            "1" : Bool;
            "2" : Bool;
            "3" : Bool;
            "4" : Bool;
            "5" : Bool;
            "6" : Bool;
            "7" : Bool;
            "8" : Bool;
            "9" : Bool;
            "10" : Bool;
            "11" : Bool;
            "12" : Bool;
            "13" : Bool;
            "14" : Bool;
            "15" : Bool;
            "16" : Bool;
         END_STRUCT;
         E_Spare_3 : Struct
            "1" : Bool;
            "2" : Bool;
            "3" : Bool;
            "4" : Bool;
            "5" : Bool;
            "6" : Bool;
            "7" : Bool;
            "8" : Bool;
            "9" : Bool;
            "10" : Bool;
            "11" : Bool;
            "12" : Bool;
            "13" : Bool;
            "14" : Bool;
            "15" : Bool;
            "16" : Bool;
         END_STRUCT;
      END_STRUCT;
      F : Struct   // RFID错误
         Robot_1 : Struct
            Grip1Error : Bool;
            Grip2Error : Bool;
            Grip1SensorCheckError : Bool;
            Grip2SensorCheckError : Bool;
            ManualMoved : Bool;
            "EXT Fault" : Bool;
            RobotNOTStart : Bool;
            "8" : Bool;
            "9" : Bool;
            "10" : Bool;
            "11" : Bool;
            "12" : Bool;
            "13" : Bool;
            "14" : Bool;
            "15" : Bool;
            "16" : Bool;
         END_STRUCT;
         Robot_2 : Struct
            Grip1Error : Bool;
            Grip2Error : Bool;
            Grip1SensorCheckError : Bool;
            Grip2SensorCheckError : Bool;
            ManualMoved : Bool;
            ReadNG_1 : Bool;
            ReadNG_2 : Bool;
            ReadNG_3 : Bool;
            ReadNG_4 : Bool;
            "EXT Fault" : Bool;
            RobotNOTStart : Bool;
            "12" : Bool;
            "13" : Bool;
            "14" : Bool;
            "15" : Bool;
            "16" : Bool;
         END_STRUCT;
         Robot_3 : Struct
            Grip1Error : Bool;
            Grip2Error : Bool;
            Grip1SensorCheckError : Bool;
            Grip2SensorCheckError : Bool;
            ManualMoved : Bool;
            "EXT Fault" : Bool;
            RobotNOTStart : Bool;
            "8" : Bool;
            "9" : Bool;
            "10" : Bool;
            "11" : Bool;
            "12" : Bool;
            "13" : Bool;
            "14" : Bool;
            "15" : Bool;
            "16" : Bool;
         END_STRUCT;
         F_Spare_1 : Struct
            Scan_805A1 : Bool;
            Robot_1 : Bool;
            Robot_2 : Bool;
            Robot_3 : Bool;
            "5" : Bool;
            "6" : Bool;
            "7" : Bool;
            "8" : Bool;
            "9" : Bool;
            "10" : Bool;
            "11" : Bool;
            "12" : Bool;
            "13" : Bool;
            "14" : Bool;
            "15" : Bool;
            "16" : Bool;
         END_STRUCT;
         F_Spare_2 : Struct
            "1" : Bool;
            "2" : Bool;
            "3" : Bool;
            "4" : Bool;
            "5" : Bool;
            "6" : Bool;
            "7" : Bool;
            "8" : Bool;
            "9" : Bool;
            "10" : Bool;
            "11" : Bool;
            "12" : Bool;
            "13" : Bool;
            "14" : Bool;
            "15" : Bool;
            "16" : Bool;
         END_STRUCT;
      END_STRUCT;
      H : Struct   // B-打标模组激光打标机1错误
         ShaftLine : Struct   // Total Error Status, Use for error code
            LiftingCylStatusError : Bool;
            LoadingStop1timeout : Bool;
            LoadingStop2timeout : Bool;
            LoadingStop3timeout : Bool;
            LoadingStop4timeout : Bool;
            UnloadingStop1timeout : Bool;
            UnloadingStop2timeout : Bool;
            UnloadingStop3timeout : Bool;
            UnloadingLiftingtimeout : Bool;
            EmptyStop1timeout : Bool;
            EmptyStop2timeout : Bool;
            EmptyStop3timeout : Bool;
            EmptyStop4timeout : Bool;
            "14" : Bool;
            "15" : Bool;
            "16" : Bool;
         END_STRUCT;
         Spare_1 : Struct
            "H-shaftLifting_Motor" : Bool;
            "H-shaftLoad_Motor" : Bool;
            "H-shaftUnLoad_Motor" : Bool;
            "4" : Bool;
            "5" : Bool;
            "6" : Bool;
            "7" : Bool;
            "8" : Bool;
            "9" : Bool;
            "10" : Bool;
            "11" : Bool;
            "12" : Bool;
            "13" : Bool;
            "14" : Bool;
            "15" : Bool;
            "16" : Bool;
         END_STRUCT;
         Spare_2 : Struct
            "1" : Bool;
            "2" : Bool;
            "3" : Bool;
            "4" : Bool;
            "5" : Bool;
            "6" : Bool;
            "7" : Bool;
            "8" : Bool;
            "9" : Bool;
            "10" : Bool;
            "11" : Bool;
            "12" : Bool;
            "13" : Bool;
            "14" : Bool;
            "15" : Bool;
            "16" : Bool;
         END_STRUCT;
         Spare_3 : Struct
            "1" : Bool;
            "2" : Bool;
            "3" : Bool;
            "4" : Bool;
            "5" : Bool;
            "6" : Bool;
            "7" : Bool;
            "8" : Bool;
            "9" : Bool;
            "10" : Bool;
            "11" : Bool;
            "12" : Bool;
            "13" : Bool;
            "14" : Bool;
            "15" : Bool;
            "16" : Bool;
         END_STRUCT;
         Spare_4 : Struct
            "1" : Bool;
            "2" : Bool;
            "3" : Bool;
            "4" : Bool;
            "5" : Bool;
            "6" : Bool;
            "7" : Bool;
            "8" : Bool;
            "9" : Bool;
            "10" : Bool;
            "11" : Bool;
            "12" : Bool;
            "13" : Bool;
            "14" : Bool;
            "15" : Bool;
            "16" : Bool;
         END_STRUCT;
      END_STRUCT;
      J : Struct
         MagnetLine : Struct   // Total Error Status, Use for error code
            LiftingCylStatusError : Bool;
            LoadingStop1timeout : Bool;
            LoadingStop2timeout : Bool;
            LoadingStop3timeout : Bool;
            LoadingStop4timeout : Bool;
            UnloadingStop1timeout : Bool;
            UnloadingStop2timeout : Bool;
            UnloadingStop3timeout : Bool;
            UnloadingLiftingtimeout : Bool;
            EmptyStop1timeout : Bool;
            EmptyStop2timeout : Bool;
            EmptyStop3timeout : Bool;
            EmptyStop4timeout : Bool;
            "14" : Bool;
            "15" : Bool;
            "16" : Bool;
         END_STRUCT;
         Spare_1 : Struct
            "J-MagnetLifting_Motor" : Bool;
            "J-MagnetLoad_Motor" : Bool;
            "J-MagnetUnLoad_Motor" : Bool;
            "4" : Bool;
            "5" : Bool;
            "6" : Bool;
            "7" : Bool;
            "8" : Bool;
            "9" : Bool;
            "10" : Bool;
            "11" : Bool;
            "12" : Bool;
            "13" : Bool;
            "14" : Bool;
            "15" : Bool;
            "16" : Bool;
         END_STRUCT;
         Spare_2 : Struct
            "1" : Bool;
            "2" : Bool;
            "3" : Bool;
            "4" : Bool;
            "5" : Bool;
            "6" : Bool;
            "7" : Bool;
            "8" : Bool;
            "9" : Bool;
            "10" : Bool;
            "11" : Bool;
            "12" : Bool;
            "13" : Bool;
            "14" : Bool;
            "15" : Bool;
            "16" : Bool;
         END_STRUCT;
         Spare_3 : Struct
            "1" : Bool;
            "2" : Bool;
            "3" : Bool;
            "4" : Bool;
            "5" : Bool;
            "6" : Bool;
            "7" : Bool;
            "8" : Bool;
            "9" : Bool;
            "10" : Bool;
            "11" : Bool;
            "12" : Bool;
            "13" : Bool;
            "14" : Bool;
            "15" : Bool;
            "16" : Bool;
         END_STRUCT;
         Spare_4 : Struct
            "1" : Bool;
            "2" : Bool;
            "3" : Bool;
            "4" : Bool;
            "5" : Bool;
            "6" : Bool;
            "7" : Bool;
            "8" : Bool;
            "9" : Bool;
            "10" : Bool;
            "11" : Bool;
            "12" : Bool;
            "13" : Bool;
            "14" : Bool;
            "15" : Bool;
            "16" : Bool;
         END_STRUCT;
      END_STRUCT;
      K : Struct
         ReserveLine : Struct   // Total Error Status, Use for error code
            LiftingCylStatusError : Bool;
            LoadingStop1timeout : Bool;
            LoadingStop2timeout : Bool;
            LoadingStop3timeout : Bool;
            LoadingStop4timeout : Bool;
            UnloadingStop1timeout : Bool;
            UnloadingStop2timeout : Bool;
            UnloadingStop3timeout : Bool;
            UnloadingLiftingtimeout : Bool;
            EmptyStop1timeout : Bool;
            EmptyStop2timeout : Bool;
            EmptyStop3timeout : Bool;
            EmptyStop4timeout : Bool;
            "14" : Bool;
            "15" : Bool;
            "16" : Bool;
         END_STRUCT;
         Spare_1 : Struct
            "K-Lifting_Motor" : Bool;
            "K-ReserveLoad_Motor" : Bool;
            "K-ReserveUnLoad_Motor" : Bool;
            "4" : Bool;
            "5" : Bool;
            "6" : Bool;
            "7" : Bool;
            "8" : Bool;
            "9" : Bool;
            "10" : Bool;
            "11" : Bool;
            "12" : Bool;
            "13" : Bool;
            "14" : Bool;
            "15" : Bool;
            "16" : Bool;
         END_STRUCT;
         Spare_2 : Struct
            "1" : Bool;
            "2" : Bool;
            "3" : Bool;
            "4" : Bool;
            "5" : Bool;
            "6" : Bool;
            "7" : Bool;
            "8" : Bool;
            "9" : Bool;
            "10" : Bool;
            "11" : Bool;
            "12" : Bool;
            "13" : Bool;
            "14" : Bool;
            "15" : Bool;
            "16" : Bool;
         END_STRUCT;
         Spare_3 : Struct
            "1" : Bool;
            "2" : Bool;
            "3" : Bool;
            "4" : Bool;
            "5" : Bool;
            "6" : Bool;
            "7" : Bool;
            "8" : Bool;
            "9" : Bool;
            "10" : Bool;
            "11" : Bool;
            "12" : Bool;
            "13" : Bool;
            "14" : Bool;
            "15" : Bool;
            "16" : Bool;
         END_STRUCT;
         Spare_4 : Struct
            "1" : Bool;
            "2" : Bool;
            "3" : Bool;
            "4" : Bool;
            "5" : Bool;
            "6" : Bool;
            "7" : Bool;
            "8" : Bool;
            "9" : Bool;
            "10" : Bool;
            "11" : Bool;
            "12" : Bool;
            "13" : Bool;
            "14" : Bool;
            "15" : Bool;
            "16" : Bool;
         END_STRUCT;
      END_STRUCT;
      L : Struct
         UnloadingLine : Struct   // Total Error Status, Use for error code
            UnloadingTransCylinderError : Bool;
            LoadingStop1timeout : Bool;
            LoadingStop2timeout : Bool;
            LoadingStop3timeout : Bool;
            LoadingStop4timeout : Bool;
            UnloadingStop1timeout : Bool;
            UnloadingStop2timeout : Bool;
            UnloadingStop3timeout : Bool;
            UnloadingLiftingtimeout : Bool;
            EmptyStop1timeout : Bool;
            EmptyStop2timeout : Bool;
            EmptyStop3timeout : Bool;
            EmptyStop4timeout : Bool;
            "14" : Bool;
            "15" : Bool;
            "16" : Bool;
         END_STRUCT;
         CuringOven : Struct
            "1" : Bool;
            "2" : Bool;
            "3" : Bool;
            "4" : Bool;
            "5" : Bool;
            "6" : Bool;
            "7" : Bool;
            "8" : Bool;
            "9" : Bool;
            "10" : Bool;
            "11" : Bool;
            "12" : Bool;
            "13" : Bool;
            "14" : Bool;
            "15" : Bool;
            "16" : Bool;
         END_STRUCT;
         Spare_2 : Struct
            "L-Unloading_Motor" : Bool;
            "L-Unloading _LineMotor" : Bool;
            "3" : Bool;
            "4" : Bool;
            "5" : Bool;
            "6" : Bool;
            "7" : Bool;
            "8" : Bool;
            "9" : Bool;
            "10" : Bool;
            "11" : Bool;
            "12" : Bool;
            "13" : Bool;
            "14" : Bool;
            "15" : Bool;
            "16" : Bool;
         END_STRUCT;
         Spare_3 : Struct
            "1" : Bool;
            "2" : Bool;
            "3" : Bool;
            "4" : Bool;
            "5" : Bool;
            "6" : Bool;
            "7" : Bool;
